Yaskawa INFORM job: N_R2_D100(P)(125,-90).JBI

/JOB
//NAME N_R2_D100(P)(125,-90)
//POS
///NPOS 515,515,515,27,0,0
///TOOL 0
///POSTYPE PULSE
///PULSE
C00000=15447,202281,164649,0,0,0
C00001=2000,202281,164649,0,0,0
C00002=24681,215512,219733,34338,41733,-28268
C00003=32295,212576,219732,43308,47198,-30665
C00004=90115,188704,203220,30079,59092,-18346
C00005=118922,140578,219095,27318,53560,2790
C00006=119744,138577,231841,24125,52341,6575
C00007=120497,123172,224477,21988,53305,9252
C00008=120847,115536,217515,22106,53618,9360
C00009=120990,112382,214541,22138,53803,9417
C00010=120986,108819,210345,21935,54503,9573
C00011=120990,112382,214541,22138,53803,9417
C00012=120993,109322,210918,21965,54414,9554
C00013=121006,109286,212535,22245,53471,9344
C00014=120993,109322,210918,21965,54414,9554
C00015=120850,112547,214017,21943,54191,9489
C00016=120501,120324,221241,21847,53796,9362
C00017=120536,123232,224555,-26557,40851,-26231
C00018=120886,115599,217598,-26179,41201,-26302
C00019=121030,112446,214627,-25996,41400,-26348
C00020=121025,108886,210434,-25635,42079,-26568
C00021=121030,112446,214627,-25996,41400,-26348
C00022=121027,109434,211061,-25684,41985,-26538
C00023=121040,109396,212675,-26172,41070,-26238
C00024=121027,109434,211061,-25684,41985,-26538
C00025=120883,112656,214154,-25882,41749,-26482
C00026=120533,120428,221368,-26294,41319,-26389
C00027=120975,122874,223899,-30521,46678,-26217
C00028=120979,115537,217604,-30470,46767,-26249
C00029=120981,112512,214915,-30422,46855,-26280
C00030=120976,108961,210733,-30079,47506,-26511
C00031=120981,112512,214915,-30422,46855,-26280
C00032=121048,109562,211421,-30089,47413,-26468
C00033=121062,109514,213024,-30551,46535,-26155
C00034=121048,109562,211421,-30089,47413,-26468
C00035=121046,112648,214220,-30153,47293,-26427
C00036=121040,120109,220750,-30241,47132,-26371
C00037=120918,149818,244976,-34417,46656,-25497
C00038=121562,167201,228013,-36113,61828,-28968
C00039=121102,161444,224515,-36573,61063,-28803
C00040=120915,159084,223008,-36750,60787,-28748
C00041=120912,155920,219969,-36672,60985,-28824
C00042=120915,159084,223008,-36750,60787,-28748
C00043=120918,156397,220402,-36676,60969,-28816
C00044=120925,157431,223143,-37055,60036,-28457
C00045=120918,156397,220402,-36676,60969,-28816
C00046=121105,158787,221971,-36508,61226,-28864
C00047=121564,164611,225614,-36067,61947,-29011
C00048=120584,167052,227666,-19839,59929,-30919
C00049=120814,161247,224144,-19904,59192,-30727
C00050=120908,158867,222626,-19923,58932,-30657
C00051=120905,155698,219577,-19875,59165,-30702
C00052=120908,158867,222626,-19923,58932,-30657
C00053=120916,156209,220066,-19878,59131,-30693
C00054=120923,157252,222817,-20111,58041,-30483
C00055=120916,156209,220066,-19878,59131,-30693
C00056=120822,158619,221647,-19864,59369,-30759
C00057=120592,164492,225315,-19810,60055,-30940
C00058=133732,167122,227890,29835,67104,20906
C00059=134129,161252,224225,30182,66361,20791
C00060=134290,158846,222649,30317,66097,20753
C00061=134272,155679,219605,30256,66314,20811
C00062=134290,158846,222649,30317,66097,20753
C00063=134298,156172,220059,30274,66286,20809
C00064=134507,157193,222762,30624,65256,20561
C00065=134298,156172,220059,30274,66286,20809
C00066=134137,158608,221700,30145,66529,20840
C00067=133740,164547,225513,29811,67224,20942
C00068=134000,188837,240725,29229,55891,39405
C00069=133801,188111,227982,27078,47780,60327
C00070=134153,183383,226108,27654,46559,60070
C00071=134296,181436,225266,27883,46096,59971
C00072=134279,178559,222861,27880,46101,59967
C00073=134296,181436,225266,27883,46096,59971
C00074=134291,178989,223219,27881,46099,59970
C00075=134475,180502,226338,28426,45044,59685
C00076=134291,178989,223219,27881,46099,59970
C00077=134148,180960,224110,27661,46546,60064
C00078=133797,185745,226100,27101,47729,60309
C00079=127590,202258,243387,866,47025,1941
C00080=121190,187961,227709,-25550,51120,-56262
C00081=120985,183329,226006,-26052,49870,-55982
C00082=120902,181420,225233,-26252,49395,-55874
C00083=120900,178540,222822,-26251,49398,-55875
C00084=120902,181420,225233,-26252,49395,-55874
C00085=120892,178980,223180,-26250,49401,-55879
C00086=120898,180522,226354,-26695,48358,-55570
C00087=120892,178980,223180,-26250,49401,-55879
C00088=120975,180912,224000,-26056,49860,-55983
C00089=121179,185599,225817,-25568,51072,-56253
C00090=121185,188297,228247,-25605,50975,-56224
C00091=120980,183661,226545,-26112,49722,-55942
C00092=120897,181750,225774,-26314,49247,-55833
C00093=120894,178874,223373,-26314,49246,-55833
C00094=120897,181750,225774,-26314,49247,-55833
C00095=120898,179301,223688,-26304,49270,-55839
C00096=120904,180831,226847,-26751,48230,-55529
C00097=120898,179301,223688,-26304,49270,-55839
C00098=120981,181234,224507,-26109,49730,-55943
C00099=121186,185925,226319,-25616,50945,-56215
C00100=123255,190595,236639,-58374,45131,30448
C00101=121545,184773,229975,-57949,45038,29555
C00102=120876,182366,227165,-57724,45033,29172
C00103=120874,179498,224782,-57730,45028,29175
C00104=120876,182366,227165,-57724,45033,29172
C00105=120862,179977,225120,-57701,45044,29152
C00106=120856,178398,221901,-56736,45697,28529
C00107=120862,179977,225120,-57701,45044,29152
C00108=121345,179993,223956,-56969,45650,28853
C00109=120328,180009,223979,-57246,45221,28671
C00110=121345,179993,223956,-56969,45650,28853
C00111=122010,182441,226833,-57205,45639,29244
C00112=123712,188347,233635,-57658,45697,30155
C00113=134995,214964,238467,-8691,44212,8832
C00114=134559,207525,231549,-8564,44604,8626
C00115=134389,204482,228633,-8506,44818,8540
C00116=134374,201971,226926,-8539,44580,8557
C00117=134389,204482,228633,-8506,44818,8540
C00118=134390,202551,227390,-8540,44593,8562
C00119=134223,200539,223898,-8355,45682,8396
C00120=134390,202551,227390,-8540,44593,8562
C00121=134560,205616,230359,-8602,44359,8650
C00122=134996,213102,237394,-8737,43918,8862
C00123=144287,210385,244112,-8132,41075,13860
C00124=162510,180487,234335,-6563,37802,23826
C00125=161591,173217,227359,-6507,38310,23477
C00126=161227,170231,224409,-6476,38572,23335
C00127=161244,167363,222022,-6476,38567,23341
C00128=161227,170231,224409,-6476,38572,23335
C00129=161271,168139,222752,-6483,38519,23354
C00130=160731,166668,219858,-6355,39511,23094
C00131=161271,168139,222752,-6483,38519,23354
C00132=161635,171154,225763,-6517,38235,23498
C00133=162555,178484,232873,-6581,37676,23852
C00134=147345,180992,237476,47268,20987,-11030
C00135=147676,173490,228422,44084,22107,-9407
C00136=147804,170370,224593,42795,22624,-8748
C00137=147814,167507,222218,42808,22614,-8751
C00138=147804,170370,224593,42795,22624,-8748
C00139=147835,168251,222850,42814,22602,-8748
C00140=147464,166660,219713,41151,23554,-8049
C00141=147835,168251,222850,42814,22602,-8748
C00142=147708,171402,226744,44147,22068,-9428
C00143=147378,178960,235933,47444,20911,-11105
C00144=133904,162048,228097,33647,50633,10192
C00145=127588,130671,218361,30951,63753,21604
C00146=128854,119558,220506,33838,57729,19894
C00147=129470,112494,214665,34247,57638,19934
C00148=129726,109579,212162,34397,57648,19967
C00149=129742,112224,215274,34604,57184,19801
C00150=129569,109596,210947,34036,58296,20180
C00151=132366,109517,211748,36018,57562,20250
C00152=135842,109408,211034,38109,57490,20655
C00153=138408,109303,210375,39617,57467,20980
C00154=138062,112231,212930,39423,57456,20929
C00155=137230,119317,218881,38897,57538,20855
C00156=115967,118809,218377,-25545,47752,-39219
C00157=116191,112195,213396,-25545,47467,-39108
C00158=116285,109468,211254,-25523,47399,-39076
C00159=116282,112131,214390,-25748,46891,-38928
C00160=116355,109459,210002,-25188,48101,-39267
C00161=118928,109470,211349,-24010,47549,-38784
C00162=122456,109452,211317,-21960,47808,-38412
C00163=125098,109423,211175,-20407,48050,-38145
C00164=124889,112154,213338,-20506,48104,-38183
C00165=124389,118775,218368,-20698,48360,-38302
C00166=123290,120857,220014,-35984,60052,-26242
C00167=122625,114409,215262,-36544,59662,-26177
C00168=122348,111754,213220,-36761,59545,-26166
C00169=122316,111747,211968,-36523,60163,-26407
C00170=122353,114378,216284,-36944,59111,-25997
C00171=119728,111769,213256,-38469,59242,-26369
C00172=117109,111771,213192,-40159,58971,-26586
C00173=123727,102355,205526,-46183,63931,-23649
C00174=124304,105056,207757,-45789,64016,-23616
C00175=125681,111582,212923,-44802,64320,-23585
C00176=122698,156476,234876,-36527,60349,-36905
C00177=122449,163722,222666,-33648,69836,-40138
C00178=121994,159688,221694,-34169,68496,-39820
C00179=121806,158013,221215,-34384,67981,-39697
C00180=121791,157173,219089,-34204,68709,-39940
C00181=121809,160369,223457,-34419,67841,-39650
C00182=120088,158037,221255,-35242,67579,-39982
C00183=118371,158016,221193,-36088,67201,-40276
C00184=122679,152032,219113,-44889,69211,-37700
C00185=123062,153728,219715,-44556,69677,-37816
C00186=123991,157822,220989,-43746,70895,-38125
C00187=117611,162371,222198,-19784,66538,-43060
C00188=117793,158216,221101,-19914,65186,-42779
C00189=117869,156493,220572,-19966,64669,-42670
C00190=117868,158864,222847,-19994,64498,-42639
C00191=117897,155666,218455,-19819,65501,-42813
C00192=119597,156527,220662,-19178,64861,-42329
C00193=121845,156504,220628,-18142,65154,-41894
C00194=123573,156435,220485,-17338,65412,-41565
C00195=123448,158166,221035,-17324,65925,-41671
C00196=123147,162343,222180,-17285,67268,-41941
C00197=130679,163960,225066,30363,74587,25346
C00198=131116,159105,222943,30757,73467,25136
C00199=131295,157106,221999,30917,73046,25058
C00200=131307,159462,224250,30949,72892,25018
C00201=131175,156320,219941,30731,73816,25246
C00202=133013,156803,221311,31804,72926,25408
C00203=135283,156324,220230,32955,72802,25889
C00204=136969,155906,219294,33795,72736,26262
C00205=136752,157909,220273,33612,73143,26338
C00206=136221,162768,222474,33163,74225,26543
C00207=131937,177942,231219,28739,51369,58836
C00208=131103,185328,225941,26199,57946,60545
C00209=131497,181762,225676,26766,56357,60246
C00210=131658,180274,225484,26999,55742,60128
C00211=131668,182419,227259,26999,55748,60133
C00212=131547,179118,223115,26715,56541,60311
C00213=133175,179856,224698,27300,55643,60570
C00214=135134,179225,223518,27660,55557,61158
C00215=136627,178672,222487,27910,55524,61620
C00216=136437,180155,222700,27670,56130,61731
C00217=135971,183707,223014,27083,57697,62015
C00218=123486,183308,222755,-21677,66267,-58163
C00219=123319,180552,223572,-22045,64449,-57850
C00220=123251,179379,223810,-22199,63739,-57726
C00221=123223,178175,221372,-22053,64554,-57898
C00222=123255,181534,225607,-22197,63742,-57725
C00223=121722,179460,223953,-22704,63409,-58082
C00224=119733,179485,223987,-23346,63019,-58556
C00225=118204,179443,223897,-23827,62749,-58927
C00226=118311,180627,223678,-23647,63452,-59052
C00227=118572,183412,222911,-23216,65258,-59366
C00228=122206,184212,222841,-27321,66765,-58270
C00229=121798,181549,223731,-27836,64961,-57929
C00230=121630,180415,223999,-28052,64257,-57793
C00231=121618,179195,221548,-27868,65037,-58001
C00232=121632,182559,225773,-28049,64266,-57795
C00233=120107,180439,224035,-28563,63890,-58140
C00234=118635,180411,223973,-29045,63559,-58483
C00235=122580,176867,224399,-39006,63999,-56229
C00236=122918,178040,224252,-38675,64647,-56380
C00237=123742,180810,223670,-37882,66314,-56760
C00238=125862,202189,241988,-26904,43300,-21160
C00239=128120,179057,235701,-24559,16531,13780
C00240=127696,171561,226511,-21973,18124,12452
C00241=127532,168433,222615,-20995,18834,11946
C00242=127606,170000,225314,-21985,18047,12432
C00243=127545,166519,221260,-21162,18697,12029
C00244=125920,168634,223016,-20023,18448,11037
C00245=112939,168466,222575,-9357,17147,2426
C00246=116539,165584,219262,-37323,21752,16959
C00247=116784,168723,223233,-38712,21158,17694
C00248=117416,176211,232564,-42212,19875,19542
C00249=121932,189645,236423,-2159,24410,9442
C00250=125769,180703,224227,31786,27614,1052
C00251=125876,172261,214331,30088,29100,1944
C00252=125917,168698,210066,29379,29784,2319
C00253=125917,170827,211817,29365,29798,2326
C00254=125970,170335,212982,30203,28938,1911
C00255=142087,161474,197407,20119,29855,11283
C00256=142171,165460,202283,20666,28944,11023
C00257=142389,174687,213323,21963,26983,10423
C00258=90115,188704,203220,30079,59092,-18346
C00259=32295,212576,219732,43308,47198,-30665
C00260=2000,202281,164649,0,0,0
C00261=15447,202281,164649,0,0,0
C00262=15447,202281,164649,0,0,0
C00263=15447,202281,164649,0,0,0
C00264=15447,202281,164649,0,0,0
C00265=-58673,196004,224446,-17944,28085,-14939
C00266=-145889,122722,224235,-48016,46095,-18882
C00267=-146704,115040,217017,-48175,46329,-19173
C00268=-147038,111863,213932,-48195,46466,-19322
C00269=-146989,108284,209714,-47640,46990,-19664
C00270=-147038,111863,213932,-48195,46466,-19322
C00271=-146995,108789,210290,-47709,46924,-19621
C00272=-147588,108743,211799,-48743,46197,-19229
C00273=-146995,108789,210290,-47709,46924,-19621
C00274=-146662,112041,213504,-47715,46759,-19455
C00275=-145849,119871,220993,-47617,46464,-19124
C00276=-145866,122721,224221,12828,42108,23463
C00277=-146680,115039,217002,12262,42622,23440
C00278=-147014,111862,213917,12020,42894,23437
C00279=-146965,108283,209699,11881,43634,23545
C00280=-147014,111862,213917,12020,42894,23437
C00281=-146966,108834,210330,11903,43530,23531
C00282=-147558,108787,211839,11788,42619,23332
C00283=-146966,108834,210330,11903,43530,23531
C00284=-146633,112084,213542,12150,43218,23530
C00285=-145821,119912,221027,12727,42616,23544
C00286=-99896,140771,234890,41057,43978,29210
C00287=-81385,119911,205689,47423,48192,34395
C00288=-80612,112172,198576,47559,48302,34669
C00289=-80295,108915,195463,47563,48400,34817
C00290=-80351,104656,190369,46930,49067,35225
C00291=-80295,108915,195463,47563,48400,34817
C00292=-80403,105399,191277,47016,48956,35141
C00293=-79657,105979,193427,48055,48085,34783
C00294=-80403,105399,191277,47016,48956,35141
C00295=-80719,108783,194591,47047,48817,34969
C00296=-81490,116767,202104,46988,48624,34642
C00297=-121434,148984,228686,40232,53743,25735
C00298=-121121,165984,226349,36450,61818,29263
C00299=-120652,160195,222770,36904,61078,29109
C00300=-120461,157820,221228,37078,60813,29058
C00301=-120460,154625,218133,36993,61025,29139
C00302=-120461,157820,221228,37078,60813,29058
C00303=-120466,155107,218575,36998,61007,29131
C00304=-120457,156175,221361,37390,60066,28768
C00305=-120466,155107,218575,36998,61007,29131
C00306=-120656,157514,220182,36833,61253,29174
C00307=-121124,163375,223912,36400,61948,29310
C00308=-120154,166157,226580,20192,59897,31174
C00309=-120372,160332,223012,20262,59178,30985
C00310=-120461,157943,221473,20283,58926,30916
C00311=-120460,154752,218385,20230,59171,30964
C00312=-120461,157943,221473,20283,58926,30916
C00313=-120471,155268,218880,20234,59135,30954
C00314=-120462,156328,221657,20479,58039,30743
C00315=-120471,155268,218880,20234,59135,30954
C00316=-120382,157688,220483,20218,59365,31019
C00317=-120164,163584,224201,20160,60032,31197
C00318=-146440,166394,227138,-35573,64457,-23044
C00319=-146979,160414,223226,-36008,63785,-22942
C00320=-147198,157963,221547,-36175,63549,-22912
C00321=-147166,154780,218475,-36088,63764,-22982
C00322=-147198,157963,221547,-36175,63549,-22912
C00323=-147192,155271,218924,-36107,63739,-22979
C00324=-147579,156256,221527,-36607,62756,-22717
C00325=-147192,155271,218924,-36107,63739,-22979
C00326=-146973,157755,220671,-35948,63955,-23001
C00327=-146435,163809,224737,-35531,64581,-23086
C00328=-120313,172340,242320,-34299,35799,-50864
C00329=-120152,166165,226604,-29898,41627,-53270
C00330=-120370,160336,223029,-30397,40891,-53053
C00331=-120459,157946,221489,-30580,40630,-52978
C00332=-120458,154754,218399,-30427,40857,-53068
C00333=-120459,157946,221489,-30580,40630,-52978
C00334=-120469,155236,218868,-30453,40819,-53057
C00335=-120460,156294,221642,-31149,39814,-52643
C00336=-120469,155236,218868,-30453,40819,-53057
C00337=-120380,157659,220474,-30285,41060,-53123
C00338=-120162,163559,224200,-29823,41748,-53319
C00339=-120808,166152,226594,30394,41466,53466
C00340=-120566,160321,223012,30904,40730,53252
C00341=-120468,157930,221468,31092,40469,53177
C00342=-120467,154738,218378,30936,40695,53270
C00343=-120468,157930,221468,31092,40469,53177
C00344=-120458,155231,218846,30958,40663,53260
C00345=-120449,156289,221621,31673,39660,52843
C00346=-120458,155231,218846,30958,40663,53260
C00347=-120556,157654,220455,30787,40904,53326
C00348=-120797,163556,224188,30312,41591,53519
C00349=-120791,196764,225758,23929,56035,57876
C00350=-120587,192763,224927,24383,54574,57590
C00351=-120504,191103,224507,24568,54012,57478
C00352=-120503,188374,222390,24597,53921,57455
C00353=-120504,191103,224507,24568,54012,57478
C00354=-120507,188771,222654,24584,53959,57464
C00355=-120500,190581,226050,24939,52900,57195
C00356=-120507,188771,222654,24584,53959,57464
C00357=-120590,190453,223116,24404,54508,57573
C00358=-120794,194507,224049,23958,55937,57852
C00359=-122901,177919,234113,63280,42164,-33162
C00360=-121117,172090,227052,62620,42118,-32100
C00361=-120421,169668,224067,62288,42131,-31644
C00362=-120420,166625,221312,62159,42195,-31566
C00363=-120421,169668,224067,62288,42131,-31644
C00364=-120408,167144,221724,62151,42197,-31556
C00365=-120417,165777,218657,61011,42789,-30863
C00366=-120408,167144,221724,62151,42197,-31556
C00367=-120925,167366,220808,61321,42738,-31237
C00368=-119855,167357,220784,61673,42315,-31065
C00369=-120925,167366,220808,61321,42738,-31237
C00370=-121617,169838,223867,61665,42707,-31701
C00371=-123392,175769,231085,62355,42716,-32781
C00372=-120775,202280,235367,5153,48165,-2931
C00373=-120574,194769,228526,5129,48504,-2846
C00374=-120495,191692,225634,5115,48698,-2809
C00375=-120494,188968,223530,5123,48593,-2814
C00376=-120495,191692,225634,5115,48698,-2809
C00377=-120503,189591,224082,5125,48574,-2818
C00378=-120509,187723,220613,5036,49745,-2759
C00379=-120503,189591,224082,5125,48574,-2818
C00380=-120581,192697,227036,5141,48357,-2856
C00381=-120782,200268,234015,5169,47964,-2945
C00382=-121097,206999,244193,5681,44142,-5775
C00383=-121079,191512,235492,5954,40481,-9245
C00384=-120657,183850,227977,5863,41145,-9051
C00385=-120492,180703,224799,5820,41473,-8971
C00386=-120490,178006,222744,5834,41353,-8978
C00387=-120492,180703,224799,5820,41473,-8971
C00388=-120494,178766,223429,5838,41322,-8982
C00389=-120501,176832,219899,5707,42495,-8905
C00390=-120494,178766,223429,5838,41322,-8982
C00391=-120660,181940,226664,5883,40972,-9064
C00392=-121082,189654,234305,5981,40258,-9262
C00393=-146775,180220,236645,-47419,21377,11449
C00394=-147132,172694,227537,-44253,22500,9822
C00395=-147271,169560,223681,-42968,23019,9160
C00396=-147281,166682,221276,-42964,23016,9155
C00397=-147271,169560,223681,-42968,23019,9160
C00398=-147302,167430,221917,-42975,23002,9154
C00399=-146946,165817,218742,-41312,23957,8448
C00400=-147302,167430,221917,-42975,23002,9154
C00401=-147164,170597,225840,-44303,22466,9837
C00402=-146807,178182,235087,-47582,21306,11517
C00403=-128844,167489,219119,15109,24995,-9484
C00404=-128455,158835,208529,13890,26957,-8768
C00405=-128304,155133,203914,13405,27852,-8482
C00406=-128303,157478,206048,13453,27746,-8505
C00407=-128377,156724,206863,13887,26890,-8745
C00408=-113473,155144,203864,7072,26584,-1170
C00409=-120204,149292,197389,35449,33024,-10735
C00410=-120464,153150,202294,36424,32253,-11330
C00411=-121134,162040,213399,38741,30633,-12744
C00412=-125965,166758,224416,9420,26881,-6319
C00413=-137280,145505,221527,-60849,19455,9531
C00414=-137453,137208,210771,-55362,20695,6872
C00415=-137521,133648,206098,-53143,21305,5791
C00416=-137716,135087,208858,-55194,20670,6709
C00417=-137560,131229,203824,-52823,21390,5626
C00418=-156550,123741,185060,-35830,21532,-8194
C00419=-156648,128309,191123,-37966,20387,-7202
C00420=-156899,138396,204316,-43383,18060,-4720
C00421=-117911,183564,223283,-22555,61467,-57170
C00422=-118076,180119,223191,-22961,59849,-56871
C00423=-118143,178678,223067,-23129,59222,-56752
C00424=-118172,177467,220617,-22939,60034,-56939
C00425=-118142,180842,224883,-23129,59217,-56751
C00426=-119670,178746,223204,-23560,58878,-57121
C00427=-121656,178756,223231,-24104,58472,-57611
C00428=-123183,178701,223135,-24507,58190,-57997
C00429=-123083,180153,223278,-24318,58813,-58115
C00430=-122836,183626,223419,-23858,60420,-58413
C00431=-123435,182649,222116,21854,66109,58333
C00432=-123257,179876,222901,22228,64300,58022
C00433=-123184,178696,223127,22385,63595,57898
C00434=-123187,180861,224942,22385,63591,57896
C00435=-123163,177487,220678,22234,64413,58071
C00436=-121656,178751,223223,22883,63276,58258
C00437=-119670,178742,223197,23516,62901,58735
C00438=-118143,178673,223059,23990,62643,59110
C00439=-118255,179863,222853,23808,63343,59234
C00440=-118526,182662,222117,23372,65138,59545
C00441=-122155,183298,221760,27476,66700,58464
C00442=-121736,180626,222622,27994,64905,58126
C00443=-121564,179487,222878,28211,64206,57992
C00444=-121566,181643,224676,28211,64207,57992
C00445=-121559,178253,220406,28022,64992,58201
C00446=-120046,179485,222867,28713,63850,58342
C00447=-118578,179431,222759,29186,63530,58689
C00448=-122506,175989,223283,39187,63899,56423
C00449=-122848,177168,223153,38856,64543,56572
C00450=-123680,179952,222608,38062,66198,56948
C00451=-122755,177840,230233,35129,68690,45019
C00452=-122402,163008,221792,33920,69743,40290
C00453=-121935,158958,220781,34447,68416,39976
C00454=-121743,157277,220286,34663,67908,39855
C00455=-121745,159644,222551,34701,67761,39805
C00456=-121735,156426,218144,34477,68638,40099
C00457=-120029,157280,220283,35512,67514,40144
C00458=-118316,157238,220178,36348,67145,40443
C00459=-122598,151300,218166,45203,69096,37849
C00460=-122985,153006,218789,44869,69556,37963
C00461=-123926,157123,220115,44056,70760,38266
C00462=-117568,161718,221460,20034,66474,43214
C00463=-117738,157551,220337,20172,65132,42934
C00464=-117808,155823,219795,20227,64620,42826
C00465=-117844,154989,217669,20075,65454,42969
C00466=-117806,158204,222092,20257,64441,42793
C00467=-119533,155877,219929,19446,64800,42481
C00468=-121779,155880,219951,18418,65078,42043
C00469=-123506,155832,219850,17618,65325,41711
C00470=-123387,157569,220410,17601,65834,41816
C00471=-123098,161760,221582,17552,67167,42086
C00472=-130606,163214,224103,-30003,74848,-25248
C00473=-131030,158350,221955,-30383,73737,-25043
C00474=-131204,156346,220999,-30538,73320,-24967
C00475=-131091,155548,218923,-30359,74095,-25155
C00476=-131214,158715,223275,-30570,73159,-24925
C00477=-132920,156060,220349,-31425,73190,-25315
C00478=-135189,155602,219317,-32580,73054,-25793
C00479=-136875,155200,218418,-33422,72979,-26163
C00480=-136662,157207,219408,-33245,73383,-26236
C00481=-136144,162078,221634,-32808,74457,-26438
C00482=-132038,149022,237746,-34581,60859,-21400
C00483=-128805,119167,220009,-33427,57827,-19835
C00484=-129404,112081,214130,-33821,57749,-19877
C00485=-129653,109155,211609,-33965,57764,-19912
C00486=-129507,109170,210390,-33615,58415,-20122
C00487=-129667,111811,214741,-34170,57293,-19745
C00488=-132294,109098,211223,-35589,57668,-20192
C00489=-135774,108996,210545,-37688,57583,-20592
C00490=-138345,108896,209914,-39203,57551,-20915
C00491=-138006,111834,212485,-39015,57535,-20863
C00492=-137190,118943,218472,-38505,57606,-20785
C00493=-115927,118422,217977,25886,47656,39303
C00494=-116133,111786,212957,25894,47383,39196
C00495=-116219,109048,210797,25875,47320,39167
C00496=-116300,109040,209546,25530,48020,39359
C00497=-116214,111722,213951,26107,46807,39015
C00498=-118862,109058,210922,24371,47459,38870
C00499=-122393,109050,210931,22328,47705,38493
C00500=-125039,109027,210818,20779,47936,38222
C00501=-124837,111767,212997,20874,47986,38258
C00502=-124356,118411,218064,21058,48232,38374
C00503=-123256,120475,219528,36367,59980,26317
C00504=-122574,114004,214729,36934,59603,26258
C00505=-122288,111339,212667,37153,59490,26250
C00506=-122292,113975,215750,37342,59054,26077
C00507=-122268,111330,211411,36904,60107,26492
C00508=-119672,111348,212674,38852,59194,26458
C00509=-117058,111342,212580,40530,58930,26680
C00510=-123636,101884,204901,46615,63860,23731
C00511=-124221,104599,207161,46219,63940,23693
C00512=-125617,111156,212391,45228,64231,23652
C00513=-58673,196004,224446,-17944,28085,-14939
C00514=15447,202281,164649,0,0,0
BC00000=0,675528,1075229
BC00001=0,1249520,1075229
BC00002=20074,1273230,1075229
BC00003=22843,1276500,1075229
BC00004=181219,1349640,881743
BC00005=259614,1271622,997019
BC00006=263455,1253369,961473
BC00007=265649,1242939,941161
BC00008=265649,1242939,941161
BC00009=265649,1242939,941161
BC00010=265649,1242939,941161
BC00011=265649,1242939,941161
BC00012=265649,1242939,941161
BC00013=265649,1242939,941161
BC00014=265649,1242939,941161
BC00015=265649,1242939,941161
BC00016=265649,1242939,941161
BC00017=279094,1259762,979345
BC00018=279094,1259762,979345
BC00019=279094,1259762,979345
BC00020=279094,1259762,979345
BC00021=279094,1259762,979345
BC00022=279094,1259762,979345
BC00023=279094,1259762,979345
BC00024=279094,1259762,979345
BC00025=279094,1259762,979345
BC00026=279094,1259762,979345
BC00027=338482,1253298,958814
BC00028=338482,1253298,958814
BC00029=338482,1253298,958814
BC00030=338482,1253298,958814
BC00031=338482,1253298,958814
BC00032=338482,1253298,958814
BC00033=338482,1253298,958814
BC00034=338482,1253298,958814
BC00035=338482,1253298,958814
BC00036=338482,1253298,958814
BC00037=333821,1266832,919202
BC00038=321005,1304050,810268
BC00039=321005,1304050,810268
BC00040=321005,1304050,810268
BC00041=321005,1304050,810268
BC00042=321005,1304050,810268
BC00043=321005,1304050,810268
BC00044=321005,1304050,810268
BC00045=321005,1304050,810268
BC00046=321005,1304050,810268
BC00047=321005,1304050,810268
BC00048=279090,1297669,836196
BC00049=279090,1297669,836196
BC00050=279090,1297669,836196
BC00051=279090,1297669,836196
BC00052=279090,1297669,836196
BC00053=279090,1297669,836196
BC00054=279090,1297669,836196
BC00055=279090,1297669,836196
BC00056=279090,1297669,836196
BC00057=279090,1297669,836196
BC00058=308990,1283728,803935
BC00059=308990,1283728,803935
BC00060=308990,1283728,803935
BC00061=308990,1283728,803935
BC00062=308990,1283728,803935
BC00063=308990,1283728,803935
BC00064=308990,1283728,803935
BC00065=308990,1283728,803935
BC00066=308990,1283728,803935
BC00067=308990,1283728,803935
BC00068=309388,1296619,799441
BC00069=309813,1310369,794648
BC00070=309813,1310369,794648
BC00071=309813,1310369,794648
BC00072=309813,1310369,794648
BC00073=309813,1310369,794648
BC00074=309813,1310369,794648
BC00075=309813,1310369,794648
BC00076=309813,1310369,794648
BC00077=309813,1310369,794648
BC00078=309813,1310369,794648
BC00079=290509,1311906,794287
BC00080=271204,1313444,793926
BC00081=271204,1313444,793926
BC00082=271204,1313444,793926
BC00083=271204,1313444,793926
BC00084=271204,1313444,793926
BC00085=271204,1313444,793926
BC00086=271204,1313444,793926
BC00087=271204,1313444,793926
BC00088=271204,1313444,793926
BC00089=271204,1313444,793926
BC00090=339752,1313535,794120
BC00091=339752,1313535,794120
BC00092=339752,1313535,794120
BC00093=339752,1313535,794120
BC00094=339752,1313535,794120
BC00095=339752,1313535,794120
BC00096=339752,1313535,794120
BC00097=339752,1313535,794120
BC00098=339752,1313535,794120
BC00099=339752,1313535,794120
BC00100=309596,1336055,723788
BC00101=309596,1336055,723788
BC00102=309596,1336055,723788
BC00103=309596,1336055,723788
BC00104=309596,1336055,723788
BC00105=309596,1336055,723788
BC00106=309596,1336055,723788
BC00107=309596,1336055,723788
BC00108=309596,1336055,723788
BC00109=309596,1336055,723788
BC00110=309596,1336055,723788
BC00111=309596,1336055,723788
BC00112=309596,1336055,723788
BC00113=366840,1349942,659049
BC00114=366840,1349942,659049
BC00115=366840,1349942,659049
BC00116=366840,1349942,659049
BC00117=366840,1349942,659049
BC00118=366840,1349942,659049
BC00119=366840,1349942,659049
BC00120=366840,1349942,659049
BC00121=366840,1349942,659049
BC00122=366840,1349942,659049
BC00123=369598,1321086,746352
BC00124=375224,1262220,924452
BC00125=375224,1262220,924452
BC00126=375224,1262220,924452
BC00127=375224,1262220,924452
BC00128=375224,1262220,924452
BC00129=375224,1262220,924452
BC00130=375224,1262220,924452
BC00131=375224,1262220,924452
BC00132=375224,1262220,924452
BC00133=375224,1262220,924452
BC00134=339925,1300732,881743
BC00135=339925,1300732,881743
BC00136=339925,1300732,881743
BC00137=339925,1300732,881743
BC00138=339925,1300732,881743
BC00139=339925,1300732,881743
BC00140=339925,1300732,881743
BC00141=339925,1300732,881743
BC00142=339925,1300732,881743
BC00143=339925,1300732,881743
BC00144=315652,1292340,901479
BC00145=299654,1262212,953023
BC00146=298993,1238691,912276
BC00147=298993,1238691,912276
BC00148=298993,1238691,912276
BC00149=298993,1238691,912276
BC00150=298993,1238691,912276
BC00151=298993,1238691,912276
BC00152=298993,1238691,912276
BC00153=298993,1238691,912276
BC00154=298993,1238691,912276
BC00155=298993,1238691,912276
BC00156=278815,1248832,951478
BC00157=278815,1248832,951478
BC00158=278815,1248832,951478
BC00159=278815,1248832,951478
BC00160=278815,1248832,951478
BC00161=278815,1248832,951478
BC00162=278815,1248832,951478
BC00163=278815,1248832,951478
BC00164=278815,1248832,951478
BC00165=278815,1248832,951478
BC00166=314804,1246682,892728
BC00167=314804,1246682,892728
BC00168=314804,1246682,892728
BC00169=314804,1246682,892728
BC00170=314804,1246682,892728
BC00171=314804,1246682,892728
BC00172=314804,1246682,892728
BC00173=314804,1246682,892728
BC00174=314804,1246682,892728
BC00175=314804,1246682,892728
BC00176=314801,1292959,892910
BC00177=314719,1294052,772836
BC00178=314719,1294052,772836
BC00179=314719,1294052,772836
BC00180=314719,1294052,772836
BC00181=314719,1294052,772836
BC00182=314719,1294052,772836
BC00183=314719,1294052,772836
BC00184=314719,1294052,772836
BC00185=314719,1294052,772836
BC00186=314719,1294052,772836
BC00187=278878,1286739,810029
BC00188=278878,1286739,810029
BC00189=278878,1286739,810029
BC00190=278878,1286739,810029
BC00191=278878,1286739,810029
BC00192=278878,1286739,810029
BC00193=278878,1286739,810029
BC00194=278878,1286739,810029
BC00195=278878,1286739,810029
BC00196=278878,1286739,810029
BC00197=311908,1275469,768683
BC00198=311908,1275469,768683
BC00199=311908,1275469,768683
BC00200=311908,1275469,768683
BC00201=311908,1275469,768683
BC00202=311908,1275469,768683
BC00203=311908,1275469,768683
BC00204=311908,1275469,768683
BC00205=311908,1275469,768683
BC00206=311908,1275469,768683
BC00207=311248,1293583,920117
BC00208=310634,1294320,778613
BC00209=310634,1294320,778613
BC00210=310634,1294320,778613
BC00211=310634,1294320,778613
BC00212=310634,1294320,778613
BC00213=310634,1294320,778613
BC00214=310634,1294320,778613
BC00215=310634,1294320,778613
BC00216=310634,1294320,778613
BC00217=310634,1294320,778613
BC00218=269571,1288878,766650
BC00219=269571,1288878,766650
BC00220=269571,1288878,766650
BC00221=269571,1288878,766650
BC00222=269571,1288878,766650
BC00223=269571,1288878,766650
BC00224=269571,1288878,766650
BC00225=269571,1288878,766650
BC00226=269571,1288878,766650
BC00227=269571,1288878,766650
BC00228=324029,1292263,751538
BC00229=324029,1292263,751538
BC00230=324029,1292263,751538
BC00231=324029,1292263,751538
BC00232=324029,1292263,751538
BC00233=324029,1292263,751538
BC00234=324029,1292263,751538
BC00235=324029,1292263,751538
BC00236=324029,1292263,751538
BC00237=324029,1292263,751538
BC00238=331457,1324273,767907
BC00239=337552,1339765,848258
BC00240=337552,1339765,848258
BC00241=337552,1339765,848258
BC00242=337552,1339765,848258
BC00243=337552,1339765,848258
BC00244=337552,1339765,848258
BC00245=337552,1339765,848258
BC00246=337552,1339765,848258
BC00247=337552,1339765,848258
BC00248=337552,1339765,848258
BC00249=326395,1340304,844891
BC00250=315775,1339017,839253
BC00251=315775,1339017,839253
BC00252=315775,1339017,839253
BC00253=315775,1339017,839253
BC00254=315775,1339017,839253
BC00255=315775,1339017,839253
BC00256=315775,1339017,839253
BC00257=315775,1339017,839253
BC00258=181219,1349640,881743
BC00259=22843,1276500,1075229
BC00260=0,1249520,1075229
BC00261=0,675528,1075229
BC00262=0,675528,1075229
BC00263=0,675528,1075229
BC00264=0,675528,1075229
BC00265=138607,763027,1056836
BC00266=322510,879121,952026
BC00267=322510,879121,952026
BC00268=322510,879121,952026
BC00269=322510,879121,952026
BC00270=322510,879121,952026
BC00271=322510,879121,952026
BC00272=322510,879121,952026
BC00273=322510,879121,952026
BC00274=322510,879121,952026
BC00275=322510,879121,952026
BC00276=326477,871688,980713
BC00277=326477,871688,980713
BC00278=326477,871688,980713
BC00279=326477,871688,980713
BC00280=326477,871688,980713
BC00281=326477,871688,980713
BC00282=326477,871688,980713
BC00283=326477,871688,980713
BC00284=326477,871688,980713
BC00285=326477,871688,980713
BC00286=267497,855485,958441
BC00287=255081,864777,953752
BC00288=255081,864777,953752
BC00289=255081,864777,953752
BC00290=255081,864777,953752
BC00291=255081,864777,953752
BC00292=255081,864777,953752
BC00293=255081,864777,953752
BC00294=255081,864777,953752
BC00295=255081,864777,953752
BC00296=255081,864777,953752
BC00297=320924,819371,961652
BC00298=320924,819371,812233
BC00299=320924,819371,812233
BC00300=320924,819371,812233
BC00301=320924,819371,812233
BC00302=320924,819371,812233
BC00303=320924,819371,812233
BC00304=320924,819371,812233
BC00305=320924,819371,812233
BC00306=320924,819371,812233
BC00307=320924,819371,812233
BC00308=278908,825639,838037
BC00309=278908,825639,838037
BC00310=278908,825639,838037
BC00311=278908,825639,838037
BC00312=278908,825639,838037
BC00313=278908,825639,838037
BC00314=278908,825639,838037
BC00315=278908,825639,838037
BC00316=278908,825639,838037
BC00317=278908,825639,838037
BC00318=344258,850073,804397
BC00319=344258,850073,804397
BC00320=344258,850073,804397
BC00321=344258,850073,804397
BC00322=344258,850073,804397
BC00323=344258,850073,804397
BC00324=344258,850073,804397
BC00325=344258,850073,804397
BC00326=344258,850073,804397
BC00327=344258,850073,804397
BC00328=268540,837164,928608
BC00329=268540,837164,928608
BC00330=268540,837164,928608
BC00331=268540,837164,928608
BC00332=268540,837164,928608
BC00333=268540,837164,928608
BC00334=268540,837164,928608
BC00335=268540,837164,928608
BC00336=268540,837164,928608
BC00337=268540,837164,928608
BC00338=268540,837164,928608
BC00339=271645,836699,929417
BC00340=271645,836699,929417
BC00341=271645,836699,929417
BC00342=271645,836699,929417
BC00343=271645,836699,929417
BC00344=271645,836699,929417
BC00345=271645,836699,929417
BC00346=271645,836699,929417
BC00347=271645,836699,929417
BC00348=271645,836699,929417
BC00349=340192,799254,723936
BC00350=340192,799254,723936
BC00351=340192,799254,723936
BC00352=340192,799254,723936
BC00353=340192,799254,723936
BC00354=340192,799254,723936
BC00355=340192,799254,723936
BC00356=340192,799254,723936
BC00357=340192,799254,723936
BC00358=340192,799254,723936
BC00359=309001,800829,792422
BC00360=309001,800829,792422
BC00361=309001,800829,792422
BC00362=309001,800829,792422
BC00363=309001,800829,792422
BC00364=309001,800829,792422
BC00365=309001,800829,792422
BC00366=309001,800829,792422
BC00367=309001,800829,792422
BC00368=309001,800829,792422
BC00369=309001,800829,792422
BC00370=309001,800829,792422
BC00371=309001,800829,792422
BC00372=321646,797982,745635
BC00373=321646,797982,745635
BC00374=321646,797982,745635
BC00375=321646,797982,745635
BC00376=321646,797982,745635
BC00377=321646,797982,745635
BC00378=321646,797982,745635
BC00379=321646,797982,745635
BC00380=321646,797982,745635
BC00381=321646,797982,745635
BC00382=296475,807012,791430
BC00383=260705,819844,856508
BC00384=260705,819844,856508
BC00385=260705,819844,856508
BC00386=260705,819844,856508
BC00387=260705,819844,856508
BC00388=260705,819844,856508
BC00389=260705,819844,856508
BC00390=260705,819844,856508
BC00391=260705,819844,856508
BC00392=260705,819844,856508
BC00393=339123,823007,883432
BC00394=339123,823007,883432
BC00395=339123,823007,883432
BC00396=339123,823007,883432
BC00397=339123,823007,883432
BC00398=339123,823007,883432
BC00399=339123,823007,883432
BC00400=339123,823007,883432
BC00401=339123,823007,883432
BC00402=339123,823007,883432
BC00403=340871,798500,921000
BC00404=340871,798500,921000
BC00405=340871,798500,921000
BC00406=340871,798500,921000
BC00407=340871,798500,921000
BC00408=340871,798500,921000
BC00409=340871,798500,921000
BC00410=340871,798500,921000
BC00411=340871,798500,921000
BC00412=343473,807454,949850
BC00413=352115,833503,1009314
BC00414=352115,833503,1009314
BC00415=352115,833503,1009314
BC00416=352115,833503,1009314
BC00417=352115,833503,1009314
BC00418=352115,833503,1009314
BC00419=352115,833503,1009314
BC00420=352115,833503,1009314
BC00421=270260,826762,778340
BC00422=270260,826762,778340
BC00423=270260,826762,778340
BC00424=270260,826762,778340
BC00425=270260,826762,778340
BC00426=270260,826762,778340
BC00427=270260,826762,778340
BC00428=270260,826762,778340
BC00429=270260,826762,778340
BC00430=270260,826762,778340
BC00431=270830,834917,768745
BC00432=270830,834917,768745
BC00433=270830,834917,768745
BC00434=270830,834917,768745
BC00435=270830,834917,768745
BC00436=270830,834917,768745
BC00437=270830,834917,768745
BC00438=270830,834917,768745
BC00439=270830,834917,768745
BC00440=270830,834917,768745
BC00441=325301,832050,753660
BC00442=325301,832050,753660
BC00443=325301,832050,753660
BC00444=325301,832050,753660
BC00445=325301,832050,753660
BC00446=325301,832050,753660
BC00447=325301,832050,753660
BC00448=325301,832050,753660
BC00449=325301,832050,753660
BC00450=325301,832050,753660
BC00451=317689,831131,771467
BC00452=315834,830096,774743
BC00453=315834,830096,774743
BC00454=315834,830096,774743
BC00455=315834,830096,774743
BC00456=315834,830096,774743
BC00457=315834,830096,774743
BC00458=315834,830096,774743
BC00459=315834,830096,774743
BC00460=315834,830096,774743
BC00461=315834,830096,774743
BC00462=279937,837039,812006
BC00463=279937,837039,812006
BC00464=279937,837039,812006
BC00465=279937,837039,812006
BC00466=279937,837039,812006
BC00467=279937,837039,812006
BC00468=279937,837039,812006
BC00469=279937,837039,812006
BC00470=279937,837039,812006
BC00471=279937,837039,812006
BC00472=312368,849486,768314
BC00473=312368,849486,768314
BC00474=312368,849486,768314
BC00475=312368,849486,768314
BC00476=312368,849486,768314
BC00477=312368,849486,768314
BC00478=312368,849486,768314
BC00479=312368,849486,768314
BC00480=312368,849486,768314
BC00481=312368,849486,768314
BC00482=304168,872987,860177
BC00483=299744,886342,911434
BC00484=299744,886342,911434
BC00485=299744,886342,911434
BC00486=299744,886342,911434
BC00487=299744,886342,911434
BC00488=299744,886342,911434
BC00489=299744,886342,911434
BC00490=299744,886342,911434
BC00491=299744,886342,911434
BC00492=299744,886342,911434
BC00493=280164,875026,952983
BC00494=280164,875026,952983
BC00495=280164,875026,952983
BC00496=280164,875026,952983
BC00497=280164,875026,952983
BC00498=280164,875026,952983
BC00499=280164,875026,952983
BC00500=280164,875026,952983
BC00501=280164,875026,952983
BC00502=280164,875026,952983
BC00503=315859,877538,894138
BC00504=315859,877538,894138
BC00505=315859,877538,894138
BC00506=315859,877538,894138
BC00507=315859,877538,894138
BC00508=315859,877538,894138
BC00509=315859,877538,894138
BC00510=315859,877538,894138
BC00511=315859,877538,894138
BC00512=315859,877538,894138
BC00513=138607,763027,1056836
BC00514=0,675528,1075229
EC00000=1108551,-556475
EC00001=1108551,-556475
EC00002=1108551,-556475
EC00003=1108551,-556475
EC00004=1108551,-556475
EC00005=1108551,-556475
EC00006=1108551,-556475
EC00007=1108551,-556475
EC00008=1108551,-556475
EC00009=1108551,-556475
EC00010=1108551,-556475
EC00011=1108551,-556475
EC00012=1108551,-556475
EC00013=1108551,-556475
EC00014=1108551,-556475
EC00015=1108551,-556475
EC00016=1108551,-556475
EC00017=1108551,-556475
EC00018=1108551,-556475
EC00019=1108551,-556475
EC00020=1108551,-556475
EC00021=1108551,-556475
EC00022=1108551,-556475
EC00023=1108551,-556475
EC00024=1108551,-556475
EC00025=1108551,-556475
EC00026=1108551,-556475
EC00027=1108551,-556475
EC00028=1108551,-556475
EC00029=1108551,-556475
EC00030=1108551,-556475
EC00031=1108551,-556475
EC00032=1108551,-556475
EC00033=1108551,-556475
EC00034=1108551,-556475
EC00035=1108551,-556475
EC00036=1108551,-556475
EC00037=1108551,-556475
EC00038=1108551,-556475
EC00039=1108551,-556475
EC00040=1108551,-556475
EC00041=1108551,-556475
EC00042=1108551,-556475
EC00043=1108551,-556475
EC00044=1108551,-556475
EC00045=1108551,-556475
EC00046=1108551,-556475
EC00047=1108551,-556475
EC00048=1108551,-556475
EC00049=1108551,-556475
EC00050=1108551,-556475
EC00051=1108551,-556475
EC00052=1108551,-556475
EC00053=1108551,-556475
EC00054=1108551,-556475
EC00055=1108551,-556475
EC00056=1108551,-556475
EC00057=1108551,-556475
EC00058=1108551,-556475
EC00059=1108551,-556475
EC00060=1108551,-556475
EC00061=1108551,-556475
EC00062=1108551,-556475
EC00063=1108551,-556475
EC00064=1108551,-556475
EC00065=1108551,-556475
EC00066=1108551,-556475
EC00067=1108551,-556475
EC00068=1108551,-556475
EC00069=1108551,-556475
EC00070=1108551,-556475
EC00071=1108551,-556475
EC00072=1108551,-556475
EC00073=1108551,-556475
EC00074=1108551,-556475
EC00075=1108551,-556475
EC00076=1108551,-556475
EC00077=1108551,-556475
EC00078=1108551,-556475
EC00079=1108551,-556475
EC00080=1108551,-556475
EC00081=1108551,-556475
EC00082=1108551,-556475
EC00083=1108551,-556475
EC00084=1108551,-556475
EC00085=1108551,-556475
EC00086=1108551,-556475
EC00087=1108551,-556475
EC00088=1108551,-556475
EC00089=1108551,-556475
EC00090=1108551,-556475
EC00091=1108551,-556475
EC00092=1108551,-556475
EC00093=1108551,-556475
EC00094=1108551,-556475
EC00095=1108551,-556475
EC00096=1108551,-556475
EC00097=1108551,-556475
EC00098=1108551,-556475
EC00099=1108551,-556475
EC00100=1108551,-556475
EC00101=1108551,-556475
EC00102=1108551,-556475
EC00103=1108551,-556475
EC00104=1108551,-556475
EC00105=1108551,-556475
EC00106=1108551,-556475
EC00107=1108551,-556475
EC00108=1108551,-556475
EC00109=1108551,-556475
EC00110=1108551,-556475
EC00111=1108551,-556475
EC00112=1108551,-556475
EC00113=1108551,-556475
EC00114=1108551,-556475
EC00115=1108551,-556475
EC00116=1108551,-556475
EC00117=1108551,-556475
EC00118=1108551,-556475
EC00119=1108551,-556475
EC00120=1108551,-556475
EC00121=1108551,-556475
EC00122=1108551,-556475
EC00123=1108551,-556475
EC00124=1108551,-556475
EC00125=1108551,-556475
EC00126=1108551,-556475
EC00127=1108551,-556475
EC00128=1108551,-556475
EC00129=1108551,-556475
EC00130=1108551,-556475
EC00131=1108551,-556475
EC00132=1108551,-556475
EC00133=1108551,-556475
EC00134=1108551,-556475
EC00135=1108551,-556475
EC00136=1108551,-556475
EC00137=1108551,-556475
EC00138=1108551,-556475
EC00139=1108551,-556475
EC00140=1108551,-556475
EC00141=1108551,-556475
EC00142=1108551,-556475
EC00143=1108551,-556475
EC00144=1108551,-556475
EC00145=1108551,-556475
EC00146=1108551,-556475
EC00147=1108551,-556475
EC00148=1108551,-556475
EC00149=1108551,-556475
EC00150=1108551,-556475
EC00151=1108551,-556475
EC00152=1108551,-556475
EC00153=1108551,-556475
EC00154=1108551,-556475
EC00155=1108551,-556475
EC00156=1108551,-556475
EC00157=1108551,-556475
EC00158=1108551,-556475
EC00159=1108551,-556475
EC00160=1108551,-556475
EC00161=1108551,-556475
EC00162=1108551,-556475
EC00163=1108551,-556475
EC00164=1108551,-556475
EC00165=1108551,-556475
EC00166=1108551,-556475
EC00167=1108551,-556475
EC00168=1108551,-556475
EC00169=1108551,-556475
EC00170=1108551,-556475
EC00171=1108551,-556475
EC00172=1108551,-556475
EC00173=1108551,-556475
EC00174=1108551,-556475
EC00175=1108551,-556475
EC00176=1108551,-556475
EC00177=1108551,-556475
EC00178=1108551,-556475
EC00179=1108551,-556475
EC00180=1108551,-556475
EC00181=1108551,-556475
EC00182=1108551,-556475
EC00183=1108551,-556475
EC00184=1108551,-556475
EC00185=1108551,-556475
EC00186=1108551,-556475
EC00187=1108551,-556475
EC00188=1108551,-556475
EC00189=1108551,-556475
EC00190=1108551,-556475
EC00191=1108551,-556475
EC00192=1108551,-556475
EC00193=1108551,-556475
EC00194=1108551,-556475
EC00195=1108551,-556475
EC00196=1108551,-556475
EC00197=1108551,-556475
EC00198=1108551,-556475
EC00199=1108551,-556475
EC00200=1108551,-556475
EC00201=1108551,-556475
EC00202=1108551,-556475
EC00203=1108551,-556475
EC00204=1108551,-556475
EC00205=1108551,-556475
EC00206=1108551,-556475
EC00207=1108551,-556475
EC00208=1108551,-556475
EC00209=1108551,-556475
EC00210=1108551,-556475
EC00211=1108551,-556475
EC00212=1108551,-556475
EC00213=1108551,-556475
EC00214=1108551,-556475
EC00215=1108551,-556475
EC00216=1108551,-556475
EC00217=1108551,-556475
EC00218=1108551,-556475
EC00219=1108551,-556475
EC00220=1108551,-556475
EC00221=1108551,-556475
EC00222=1108551,-556475
EC00223=1108551,-556475
EC00224=1108551,-556475
EC00225=1108551,-556475
EC00226=1108551,-556475
EC00227=1108551,-556475
EC00228=1108551,-556475
EC00229=1108551,-556475
EC00230=1108551,-556475
EC00231=1108551,-556475
EC00232=1108551,-556475
EC00233=1108551,-556475
EC00234=1108551,-556475
EC00235=1108551,-556475
EC00236=1108551,-556475
EC00237=1108551,-556475
EC00238=1108551,-556475
EC00239=1108551,-556475
EC00240=1108551,-556475
EC00241=1108551,-556475
EC00242=1108551,-556475
EC00243=1108551,-556475
EC00244=1108551,-556475
EC00245=1108551,-556475
EC00246=1108551,-556475
EC00247=1108551,-556475
EC00248=1108551,-556475
EC00249=1108551,-556475
EC00250=1108551,-556475
EC00251=1108551,-556475
EC00252=1108551,-556475
EC00253=1108551,-556475
EC00254=1108551,-556475
EC00255=1108551,-556475
EC00256=1108551,-556475
EC00257=1108551,-556475
EC00258=1108551,-556475
EC00259=1108551,-556475
EC00260=1108551,-556475
EC00261=1108551,-556475
EC00262=266052,-556475
EC00263=-266052,556475
EC00264=-1108551,556475
EC00265=-1108551,556475
EC00266=-1108551,556475
EC00267=-1108551,556475
EC00268=-1108551,556475
EC00269=-1108551,556475
EC00270=-1108551,556475
EC00271=-1108551,556475
EC00272=-1108551,556475
EC00273=-1108551,556475
EC00274=-1108551,556475
EC00275=-1108551,556475
EC00276=-1108551,556475
EC00277=-1108551,556475
EC00278=-1108551,556475
EC00279=-1108551,556475
EC00280=-1108551,556475
EC00281=-1108551,556475
EC00282=-1108551,556475
EC00283=-1108551,556475
EC00284=-1108551,556475
EC00285=-1108551,556475
EC00286=-1108551,556475
EC00287=-1108551,556475
EC00288=-1108551,556475
EC00289=-1108551,556475
EC00290=-1108551,556475
EC00291=-1108551,556475
EC00292=-1108551,556475
EC00293=-1108551,556475
EC00294=-1108551,556475
EC00295=-1108551,556475
EC00296=-1108551,556475
EC00297=-1108551,556475
EC00298=-1108551,556475
EC00299=-1108551,556475
EC00300=-1108551,556475
EC00301=-1108551,556475
EC00302=-1108551,556475
EC00303=-1108551,556475
EC00304=-1108551,556475
EC00305=-1108551,556475
EC00306=-1108551,556475
EC00307=-1108551,556475
EC00308=-1108551,556475
EC00309=-1108551,556475
EC00310=-1108551,556475
EC00311=-1108551,556475
EC00312=-1108551,556475
EC00313=-1108551,556475
EC00314=-1108551,556475
EC00315=-1108551,556475
EC00316=-1108551,556475
EC00317=-1108551,556475
EC00318=-1108551,556475
EC00319=-1108551,556475
EC00320=-1108551,556475
EC00321=-1108551,556475
EC00322=-1108551,556475
EC00323=-1108551,556475
EC00324=-1108551,556475
EC00325=-1108551,556475
EC00326=-1108551,556475
EC00327=-1108551,556475
EC00328=-1108551,556475
EC00329=-1108551,556475
EC00330=-1108551,556475
EC00331=-1108551,556475
EC00332=-1108551,556475
EC00333=-1108551,556475
EC00334=-1108551,556475
EC00335=-1108551,556475
EC00336=-1108551,556475
EC00337=-1108551,556475
EC00338=-1108551,556475
EC00339=-1108551,556475
EC00340=-1108551,556475
EC00341=-1108551,556475
EC00342=-1108551,556475
EC00343=-1108551,556475
EC00344=-1108551,556475
EC00345=-1108551,556475
EC00346=-1108551,556475
EC00347=-1108551,556475
EC00348=-1108551,556475
EC00349=-1108551,556475
EC00350=-1108551,556475
EC00351=-1108551,556475
EC00352=-1108551,556475
EC00353=-1108551,556475
EC00354=-1108551,556475
EC00355=-1108551,556475
EC00356=-1108551,556475
EC00357=-1108551,556475
EC00358=-1108551,556475
EC00359=-1108551,556475
EC00360=-1108551,556475
EC00361=-1108551,556475
EC00362=-1108551,556475
EC00363=-1108551,556475
EC00364=-1108551,556475
EC00365=-1108551,556475
EC00366=-1108551,556475
EC00367=-1108551,556475
EC00368=-1108551,556475
EC00369=-1108551,556475
EC00370=-1108551,556475
EC00371=-1108551,556475
EC00372=-1108551,556475
EC00373=-1108551,556475
EC00374=-1108551,556475
EC00375=-1108551,556475
EC00376=-1108551,556475
EC00377=-1108551,556475
EC00378=-1108551,556475
EC00379=-1108551,556475
EC00380=-1108551,556475
EC00381=-1108551,556475
EC00382=-1108551,556475
EC00383=-1108551,556475
EC00384=-1108551,556475
EC00385=-1108551,556475
EC00386=-1108551,556475
EC00387=-1108551,556475
EC00388=-1108551,556475
EC00389=-1108551,556475
EC00390=-1108551,556475
EC00391=-1108551,556475
EC00392=-1108551,556475
EC00393=-1108551,556475
EC00394=-1108551,556475
EC00395=-1108551,556475
EC00396=-1108551,556475
EC00397=-1108551,556475
EC00398=-1108551,556475
EC00399=-1108551,556475
EC00400=-1108551,556475
EC00401=-1108551,556475
EC00402=-1108551,556475
EC00403=-1108551,556475
EC00404=-1108551,556475
EC00405=-1108551,556475
EC00406=-1108551,556475
EC00407=-1108551,556475
EC00408=-1108551,556475
EC00409=-1108551,556475
EC00410=-1108551,556475
EC00411=-1108551,556475
EC00412=-1108551,556475
EC00413=-1108551,556475
EC00414=-1108551,556475
EC00415=-1108551,556475
EC00416=-1108551,556475
EC00417=-1108551,556475
EC00418=-1108551,556475
EC00419=-1108551,556475
EC00420=-1108551,556475
EC00421=-1108551,556475
EC00422=-1108551,556475
EC00423=-1108551,556475
EC00424=-1108551,556475
EC00425=-1108551,556475
EC00426=-1108551,556475
EC00427=-1108551,556475
EC00428=-1108551,556475
EC00429=-1108551,556475
EC00430=-1108551,556475
EC00431=-1108551,556475
EC00432=-1108551,556475
EC00433=-1108551,556475
EC00434=-1108551,556475
EC00435=-1108551,556475
EC00436=-1108551,556475
EC00437=-1108551,556475
EC00438=-1108551,556475
EC00439=-1108551,556475
EC00440=-1108551,556475
EC00441=-1108551,556475
EC00442=-1108551,556475
EC00443=-1108551,556475
EC00444=-1108551,556475
EC00445=-1108551,556475
EC00446=-1108551,556475
EC00447=-1108551,556475
EC00448=-1108551,556475
EC00449=-1108551,556475
EC00450=-1108551,556475
EC00451=-1108551,556475
EC00452=-1108551,556475
EC00453=-1108551,556475
EC00454=-1108551,556475
EC00455=-1108551,556475
EC00456=-1108551,556475
EC00457=-1108551,556475
EC00458=-1108551,556475
EC00459=-1108551,556475
EC00460=-1108551,556475
EC00461=-1108551,556475
EC00462=-1108551,556475
EC00463=-1108551,556475
EC00464=-1108551,556475
EC00465=-1108551,556475
EC00466=-1108551,556475
EC00467=-1108551,556475
EC00468=-1108551,556475
EC00469=-1108551,556475
EC00470=-1108551,556475
EC00471=-1108551,556475
EC00472=-1108551,556475
EC00473=-1108551,556475
EC00474=-1108551,556475
EC00475=-1108551,556475
EC00476=-1108551,556475
EC00477=-1108551,556475
EC00478=-1108551,556475
EC00479=-1108551,556475
EC00480=-1108551,556475
EC00481=-1108551,556475
EC00482=-1108551,556475
EC00483=-1108551,556475
EC00484=-1108551,556475
EC00485=-1108551,556475
EC00486=-1108551,556475
EC00487=-1108551,556475
EC00488=-1108551,556475
EC00489=-1108551,556475
EC00490=-1108551,556475
EC00491=-1108551,556475
EC00492=-1108551,556475
EC00493=-1108551,556475
EC00494=-1108551,556475
EC00495=-1108551,556475
EC00496=-1108551,556475
EC00497=-1108551,556475
EC00498=-1108551,556475
EC00499=-1108551,556475
EC00500=-1108551,556475
EC00501=-1108551,556475
EC00502=-1108551,556475
EC00503=-1108551,556475
EC00504=-1108551,556475
EC00505=-1108551,556475
EC00506=-1108551,556475
EC00507=-1108551,556475
EC00508=-1108551,556475
EC00509=-1108551,556475
EC00510=-1108551,556475
EC00511=-1108551,556475
EC00512=-1108551,556475
EC00513=-1108551,556475
EC00514=-1108551,556475
///POSTYPE BASE
///RECTAN
///RCONF 0,0,0,0,0,0,0,0,0,0,0,0,0,0,0,0,0,0,0,0,0,0,0,0
P00006=0.222,-3.123,-1.508,0.0000,0.0000,0.0000
P00021=-0.225,-6.128,-0.405,0.0000,0.0000,0.0000
P00022=0.222,-3.123,-1.508,0.0000,0.0000,0.0000
P00023=0.143,-0.036,0.682,0.0000,0.0000,0.0000
P00024=0.145,-0.552,1.326,0.0000,0.0000,0.0000
P00025=-2.003,0.006,0.728,0.0000,0.0000,0.0000
P00026=0.562,-0.002,-0.337,0.0000,0.0000,0.0000
P00027=-0.746,0.015,-9.096,0.0000,0.0000,0.0000
P00028=-2.237,-0.018,-7.702,0.0000,0.0000,0.0000
P00029=-2.156,-0.086,-4.681,0.0000,0.0000,0.0000
P00030=5.926,-4.294,-1.390,0.0000,0.0000,0.0000
P00031=1.853,-0.001,-1.549,0.0000,0.0000,0.0000
P00032=1.957,0.503,-7.217,0.0000,0.0000,0.0000
///RCONF 0,0,0,0,1,0,0,0,0,0,0,0,0,0,0,0,0,0,0,0,0,0,0,0
P00033=-0.123,0.612,-5.012,0.0000,0.0000,0.0000
///RCONF 0,0,0,0,0,0,0,0,0,0,0,0,0,0,0,0,0,0,0,0,0,0,0,0
P00041=0.192,3.924,0.305,0.0000,0.0000,0.0000
P00042=-0.217,1.941,0.413,0.0000,0.0000,0.0000
P00043=-0.044,-1.937,1.197,0.0000,0.0000,0.0000
P00044=0.687,-2.322,1.156,0.0000,0.0000,0.0000
P00045=-0.068,-0.810,1.603,0.0000,0.0000,0.0000
P00046=0.799,0.043,1.292,0.0000,0.0000,0.0000
///RCONF 0,1,0,0,0,0,0,0,0,0,0,0,0,0,0,0,0,0,0,0,0,0,0,0
P00047=-0.011,1.737,-0.646,0.0000,0.0000,0.0000
///RCONF 0,0,0,0,0,0,0,0,0,0,0,0,0,0,0,0,0,0,0,0,0,0,0,0
P00048=2.411,0.025,-0.606,0.0000,0.0000,0.0000
P00049=3.413,-3.572,-1.618,0.0000,0.0000,0.0000
P00050=4.296,-4.501,-0.826,0.0000,0.0000,0.0000
P00051=0.367,3.892,0.009,0.0000,0.0000,0.0000
P00052=0.088,2.832,-0.342,0.0000,0.0000,0.0000
P00053=0.134,6.594,0.107,0.0000,0.0000,0.0000
//INST
///DATE 2024/02/02 10:05
///ATTR SC,RW
///GROUP1 RB1,BS1
///GROUP2 ST1
NOP
'N_r2_D100(P)(125,-90)
'
MOVJ C00000 BC00000 VJ=100.00  +MOVJ EC00000 VJ=100.00
MOVJ C00001 BC00001 VJ=100.00  +MOVJ EC00001 VJ=100.00
'
MOVJ C00002 BC00002 VJ=100.00  +MOVJ EC00002 VJ=100.00
MOVJ C00003 BC00003 VJ=100.00  +MOVJ EC00003 VJ=100.00
MOVJ C00004 BC00004 VJ=100.00  +MOVJ EC00004 VJ=100.00
MOVJ C00005 BC00005 VJ=100.00  +MOVJ EC00005 VJ=100.00
MOVJ C00006 BC00006 VJ=100.00  +MOVJ EC00006 VJ=100.00
'Path S3336
SSFTOF
MOVJ C00007 BC00007 VJ=100.00  +MOVJ EC00007 VJ=100.00
MOVL C00008 BC00008 V=400.0  +MOVJ EC00008 VJ=100.00
SMOVL C00009 BC00009 V=100.0  +MOVJ EC00009
SREFP 3 C00010 BC00010  +REFP EC00010
CALL JOB:SEARCH-R1-S1
SET P021 P006
SSFTON P021
SMOVL C00011 BC00011 V=100.0  +MOVJ EC00011
SMOVL C00012 BC00012 V=100.0  +MOVJ EC00012
SREFP 3 C00013 BC00013  +REFP EC00013
CALL JOB:SEARCH-R1-S1
SET P021 P006
SSFTON P021
SMOVL C00014 BC00014 V=100.0  +MOVJ EC00014
MOVL C00015 BC00015 V=400.0  +MOVJ EC00015 VJ=100.00
MOVL C00016 BC00016 V=1000.0  +MOVJ EC00016 VJ=100.00
'Path S3337
SSFTOF
MOVJ C00017 BC00017 VJ=100.00  +MOVJ EC00017 VJ=100.00
MOVL C00018 BC00018 V=400.0  +MOVJ EC00018 VJ=100.00
SMOVL C00019 BC00019 V=100.0  +MOVJ EC00019
SREFP 3 C00020 BC00020  +REFP EC00020
CALL JOB:SEARCH-R1-S1
SET P022 P006
SSFTON P022
SMOVL C00021 BC00021 V=100.0  +MOVJ EC00021
SMOVL C00022 BC00022 V=100.0  +MOVJ EC00022
SREFP 3 C00023 BC00023  +REFP EC00023
CALL JOB:SEARCH-R1-S1
SET P022 P006
SSFTON P022
SMOVL C00024 BC00024 V=100.0  +MOVJ EC00024
MOVL C00025 BC00025 V=400.0  +MOVJ EC00025 VJ=100.00
MOVL C00026 BC00026 V=1000.0  +MOVJ EC00026 VJ=100.00
'Path S3338
SSFTOF
MOVJ C00027 BC00027 VJ=100.00  +MOVJ EC00027 VJ=100.00
MOVL C00028 BC00028 V=400.0  +MOVJ EC00028 VJ=100.00
SMOVL C00029 BC00029 V=100.0  +MOVJ EC00029
SREFP 3 C00030 BC00030  +REFP EC00030
CALL JOB:SEARCH-R1-S1
SET P023 P006
SSFTON P023
SMOVL C00031 BC00031 V=100.0  +MOVJ EC00031
SMOVL C00032 BC00032 V=100.0  +MOVJ EC00032
SREFP 3 C00033 BC00033  +REFP EC00033
CALL JOB:SEARCH-R1-S1
SET P023 P006
SSFTON P023
SMOVL C00034 BC00034 V=100.0  +MOVJ EC00034
MOVL C00035 BC00035 V=400.0  +MOVJ EC00035 VJ=100.00
MOVL C00036 BC00036 V=1000.0  +MOVJ EC00036 VJ=100.00
MOVJ C00037 BC00037 VJ=100.00  +MOVJ EC00037 VJ=100.00
'Path S3339
SSFTOF
MOVJ C00038 BC00038 VJ=100.00  +MOVJ EC00038 VJ=100.00
MOVL C00039 BC00039 V=400.0  +MOVJ EC00039 VJ=100.00
SMOVL C00040 BC00040 V=100.0  +MOVJ EC00040
SREFP 3 C00041 BC00041  +REFP EC00041
CALL JOB:SEARCH-R1-S1
SET P024 P006
SSFTON P024
SMOVL C00042 BC00042 V=100.0  +MOVJ EC00042
SMOVL C00043 BC00043 V=100.0  +MOVJ EC00043
SREFP 3 C00044 BC00044  +REFP EC00044
CALL JOB:SEARCH-R1-S1
SET P024 P006
SSFTON P024
SMOVL C00045 BC00045 V=100.0  +MOVJ EC00045
MOVL C00046 BC00046 V=400.0  +MOVJ EC00046 VJ=100.00
MOVL C00047 BC00047 V=1000.0  +MOVJ EC00047 VJ=100.00
'Path S3341
SSFTOF
MOVJ C00048 BC00048 VJ=100.00  +MOVJ EC00048 VJ=100.00
MOVL C00049 BC00049 V=400.0  +MOVJ EC00049 VJ=100.00
SMOVL C00050 BC00050 V=100.0  +MOVJ EC00050
SREFP 3 C00051 BC00051  +REFP EC00051
CALL JOB:SEARCH-R1-S1
SET P025 P006
SSFTON P025
SMOVL C00052 BC00052 V=100.0  +MOVJ EC00052
SMOVL C00053 BC00053 V=100.0  +MOVJ EC00053
SREFP 3 C00054 BC00054  +REFP EC00054
CALL JOB:SEARCH-R1-S1
SET P025 P006
SSFTON P025
SMOVL C00055 BC00055 V=100.0  +MOVJ EC00055
MOVL C00056 BC00056 V=400.0  +MOVJ EC00056 VJ=100.00
MOVL C00057 BC00057 V=1000.0  +MOVJ EC00057 VJ=100.00
'Path S3343
SSFTOF
MOVJ C00058 BC00058 VJ=100.00  +MOVJ EC00058 VJ=100.00
MOVL C00059 BC00059 V=400.0  +MOVJ EC00059 VJ=100.00
SMOVL C00060 BC00060 V=100.0  +MOVJ EC00060
SREFP 3 C00061 BC00061  +REFP EC00061
CALL JOB:SEARCH-R1-S1
SET P026 P006
SSFTON P026
SMOVL C00062 BC00062 V=100.0  +MOVJ EC00062
SMOVL C00063 BC00063 V=100.0  +MOVJ EC00063
SREFP 3 C00064 BC00064  +REFP EC00064
CALL JOB:SEARCH-R1-S1
SET P026 P006
SSFTON P026
SMOVL C00065 BC00065 V=100.0  +MOVJ EC00065
MOVL C00066 BC00066 V=400.0  +MOVJ EC00066 VJ=100.00
MOVL C00067 BC00067 V=1000.0  +MOVJ EC00067 VJ=100.00
MOVJ C00068 BC00068 VJ=100.00  +MOVJ EC00068 VJ=100.00
'Path S3345
SSFTOF
MOVJ C00069 BC00069 VJ=100.00  +MOVJ EC00069 VJ=100.00
MOVL C00070 BC00070 V=400.0  +MOVJ EC00070 VJ=100.00
SMOVL C00071 BC00071 V=100.0  +MOVJ EC00071
SREFP 3 C00072 BC00072  +REFP EC00072
CALL JOB:SEARCH-R1-S1
SET P027 P006
SSFTON P027
SMOVL C00073 BC00073 V=100.0  +MOVJ EC00073
SMOVL C00074 BC00074 V=100.0  +MOVJ EC00074
SREFP 3 C00075 BC00075  +REFP EC00075
CALL JOB:SEARCH-R1-S1
SET P027 P006
SSFTON P027
SMOVL C00076 BC00076 V=100.0  +MOVJ EC00076
MOVL C00077 BC00077 V=400.0  +MOVJ EC00077 VJ=100.00
MOVL C00078 BC00078 V=1000.0  +MOVJ EC00078 VJ=100.00
MOVJ C00079 BC00079 VJ=100.00  +MOVJ EC00079 VJ=100.00
'Path S3347
SSFTOF
MOVJ C00080 BC00080 VJ=100.00  +MOVJ EC00080 VJ=100.00
MOVL C00081 BC00081 V=400.0  +MOVJ EC00081 VJ=100.00
SMOVL C00082 BC00082 V=100.0  +MOVJ EC00082
SREFP 3 C00083 BC00083  +REFP EC00083
CALL JOB:SEARCH-R1-S1
SET P028 P006
SSFTON P028
SMOVL C00084 BC00084 V=100.0  +MOVJ EC00084
SMOVL C00085 BC00085 V=100.0  +MOVJ EC00085
SREFP 3 C00086 BC00086  +REFP EC00086
CALL JOB:SEARCH-R1-S1
SET P028 P006
SSFTON P028
SMOVL C00087 BC00087 V=100.0  +MOVJ EC00087
MOVL C00088 BC00088 V=400.0  +MOVJ EC00088 VJ=100.00
MOVL C00089 BC00089 V=1000.0  +MOVJ EC00089 VJ=100.00
'Path S3349
SSFTOF
MOVJ C00090 BC00090 VJ=100.00  +MOVJ EC00090 VJ=100.00
MOVL C00091 BC00091 V=400.0  +MOVJ EC00091 VJ=100.00
SMOVL C00092 BC00092 V=100.0  +MOVJ EC00092
SREFP 3 C00093 BC00093  +REFP EC00093
CALL JOB:SEARCH-R1-S1
SET P029 P006
SSFTON P029
SMOVL C00094 BC00094 V=100.0  +MOVJ EC00094
SMOVL C00095 BC00095 V=100.0  +MOVJ EC00095
SREFP 3 C00096 BC00096  +REFP EC00096
CALL JOB:SEARCH-R1-S1
SET P029 P006
SSFTON P029
SMOVL C00097 BC00097 V=100.0  +MOVJ EC00097
MOVL C00098 BC00098 V=400.0  +MOVJ EC00098 VJ=100.00
MOVL C00099 BC00099 V=1000.0  +MOVJ EC00099 VJ=100.00
'Path S3350
SSFTOF
MOVJ C00100 BC00100 VJ=100.00  +MOVJ EC00100 VJ=100.00
MOVL C00101 BC00101 V=400.0  +MOVJ EC00101 VJ=100.00
SMOVL C00102 BC00102 V=100.0  +MOVJ EC00102
SREFP 3 C00103 BC00103  +REFP EC00103
CALL JOB:SEARCH-R1-S1
SET P030 P006
SSFTON P030
SMOVL C00104 BC00104 V=100.0  +MOVJ EC00104
SMOVL C00105 BC00105 V=100.0  +MOVJ EC00105
SREFP 3 C00106 BC00106  +REFP EC00106
CALL JOB:SEARCH-R1-S1
SET P030 P006
SSFTON P030
SMOVL C00107 BC00107 V=100.0  +MOVJ EC00107
SMOVL C00108 BC00108 V=100.0  +MOVJ EC00108
SREFP 3 C00109 BC00109  +REFP EC00109
CALL JOB:SEARCH-R1-S1
SET P030 P006
SSFTON P030
SMOVL C00110 BC00110 V=100.0  +MOVJ EC00110
MOVL C00111 BC00111 V=400.0  +MOVJ EC00111 VJ=100.00
MOVL C00112 BC00112 V=1000.0  +MOVJ EC00112 VJ=100.00
'Path S3351
SSFTOF
MOVJ C00113 BC00113 VJ=100.00  +MOVJ EC00113 VJ=100.00
MOVL C00114 BC00114 V=400.0  +MOVJ EC00114 VJ=100.00
SMOVL C00115 BC00115 V=100.0  +MOVJ EC00115
SREFP 3 C00116 BC00116  +REFP EC00116
CALL JOB:SEARCH-R1-S1
SET P031 P006
SSFTON P031
SMOVL C00117 BC00117 V=100.0  +MOVJ EC00117
SMOVL C00118 BC00118 V=100.0  +MOVJ EC00118
SREFP 3 C00119 BC00119  +REFP EC00119
CALL JOB:SEARCH-R1-S1
SET P031 P006
SSFTON P031
SMOVL C00120 BC00120 V=100.0  +MOVJ EC00120
MOVL C00121 BC00121 V=400.0  +MOVJ EC00121 VJ=100.00
MOVL C00122 BC00122 V=1000.0  +MOVJ EC00122 VJ=100.00
MOVJ C00123 BC00123 VJ=100.00  +MOVJ EC00123 VJ=100.00
'Path S3352
SSFTOF
MOVJ C00124 BC00124 VJ=100.00  +MOVJ EC00124 VJ=100.00
MOVL C00125 BC00125 V=400.0  +MOVJ EC00125 VJ=100.00
SMOVL C00126 BC00126 V=100.0  +MOVJ EC00126
SREFP 3 C00127 BC00127  +REFP EC00127
CALL JOB:SEARCH-R1-S1
SET P032 P006
SSFTON P032
SMOVL C00128 BC00128 V=100.0  +MOVJ EC00128
SMOVL C00129 BC00129 V=100.0  +MOVJ EC00129
SREFP 3 C00130 BC00130  +REFP EC00130
CALL JOB:SEARCH-R1-S1
SET P032 P006
SSFTON P032
SMOVL C00131 BC00131 V=100.0  +MOVJ EC00131
MOVL C00132 BC00132 V=400.0  +MOVJ EC00132 VJ=100.00
MOVL C00133 BC00133 V=1000.0  +MOVJ EC00133 VJ=100.00
'Path S3353
SSFTOF
MOVJ C00134 BC00134 VJ=100.00  +MOVJ EC00134 VJ=100.00
MOVL C00135 BC00135 V=400.0  +MOVJ EC00135 VJ=100.00
SMOVL C00136 BC00136 V=100.0  +MOVJ EC00136
SREFP 3 C00137 BC00137  +REFP EC00137
CALL JOB:SEARCH-R1-S1
SET P033 P006
SSFTON P033
SMOVL C00138 BC00138 V=100.0  +MOVJ EC00138
SMOVL C00139 BC00139 V=100.0  +MOVJ EC00139
SREFP 3 C00140 BC00140  +REFP EC00140
CALL JOB:SEARCH-R1-S1
SET P033 P006
SSFTON P033
SMOVL C00141 BC00141 V=100.0  +MOVJ EC00141
MOVL C00142 BC00142 V=400.0  +MOVJ EC00142 VJ=100.00
MOVL C00143 BC00143 V=1000.0  +MOVJ EC00143 VJ=100.00
MOVJ C00144 BC00144 VJ=100.00  +MOVJ EC00144 VJ=100.00
MOVJ C00145 BC00145 VJ=100.00  +MOVJ EC00145 VJ=100.00
'Path W3292
SSFTOF
SSFTON P021
MOVJ C00146 BC00146 VJ=100.00  +MOVJ EC00146 VJ=100.00
SMOVL C00147 BC00147 V=400.0  +MOVJ EC00147
SMOVL C00148 BC00148 V=100.0 PL=0  +MOVJ EC00148
SREFP 1 C00149 BC00149  +REFP EC00149
SREFP 2 C00150 BC00150  +REFP EC00150
MACRO1 MJ#(0) ARGF0
ARCON
SMOVL C00151 BC00151 V=10.0  +MOVJ EC00151
SMOVL C00152 BC00152 V=10.0  +MOVJ EC00152
SMOVL C00153 BC00153 V=10.0  +MOVJ EC00153
ARCOF
SMOVL C00154 BC00154 V=400.0  +MOVJ EC00154
SMOVL C00155 BC00155 V=1000.0  +MOVJ EC00155
SSFTOF
'Path W3293
SSFTOF
SSFTON P022
MOVJ C00156 BC00156 VJ=100.00  +MOVJ EC00156 VJ=100.00
SMOVL C00157 BC00157 V=400.0  +MOVJ EC00157
SMOVL C00158 BC00158 V=100.0 PL=0  +MOVJ EC00158
SREFP 1 C00159 BC00159  +REFP EC00159
SREFP 2 C00160 BC00160  +REFP EC00160
MACRO1 MJ#(0) ARGF0
ARCON
SMOVL C00161 BC00161 V=10.0  +MOVJ EC00161
SMOVL C00162 BC00162 V=10.0  +MOVJ EC00162
SMOVL C00163 BC00163 V=10.0  +MOVJ EC00163
ARCOF
SMOVL C00164 BC00164 V=400.0  +MOVJ EC00164
SMOVL C00165 BC00165 V=1000.0  +MOVJ EC00165
SSFTOF
'Path W3294
SSFTOF
SSFTON P023
MOVJ C00166 BC00166 VJ=100.00  +MOVJ EC00166 VJ=100.00
SMOVL C00167 BC00167 V=400.0  +MOVJ EC00167
SMOVL C00168 BC00168 V=100.0 PL=0  +MOVJ EC00168
SREFP 1 C00169 BC00169  +REFP EC00169
SREFP 2 C00170 BC00170  +REFP EC00170
MACRO1 MJ#(0) ARGF0
ARCON
SMOVL C00171 BC00171 V=10.0  +MOVJ EC00171
SMOVL C00172 BC00172 V=10.0  +MOVJ EC00172
SMOVL C00173 BC00173 V=10.0  +MOVJ EC00173
ARCOF
SMOVL C00174 BC00174 V=400.0  +MOVJ EC00174
SMOVL C00175 BC00175 V=1000.0  +MOVJ EC00175
SSFTOF
'
MOVJ C00176 BC00176 VJ=100.00  +MOVJ EC00176 VJ=100.00
'Path W3340
SSFTOF
SSFTON P024
MOVJ C00177 BC00177 VJ=100.00  +MOVJ EC00177 VJ=100.00
SMOVL C00178 BC00178 V=400.0  +MOVJ EC00178
SMOVL C00179 BC00179 V=150.0 PL=0  +MOVJ EC00179
SREFP 1 C00180 BC00180  +REFP EC00180
SREFP 2 C00181 BC00181  +REFP EC00181
MACRO1 MJ#(0) ARGF0
ARCON
SMOVL C00182 BC00182 V=10.0  +MOVJ EC00182
SMOVL C00183 BC00183 V=10.0  +MOVJ EC00183
SMOVL C00184 BC00184 V=10.0  +MOVJ EC00184
ARCOF
SMOVL C00185 BC00185 V=400.0  +MOVJ EC00185
SMOVL C00186 BC00186 V=1000.0  +MOVJ EC00186
SSFTOF
'Path W3342
SSFTOF
SSFTON P025
MOVJ C00187 BC00187 VJ=100.00  +MOVJ EC00187 VJ=100.00
SMOVL C00188 BC00188 V=400.0  +MOVJ EC00188
SMOVL C00189 BC00189 V=150.0 PL=0  +MOVJ EC00189
SREFP 1 C00190 BC00190  +REFP EC00190
SREFP 2 C00191 BC00191  +REFP EC00191
MACRO1 MJ#(0) ARGF0
ARCON
SMOVL C00192 BC00192 V=10.0  +MOVJ EC00192
SMOVL C00193 BC00193 V=10.0  +MOVJ EC00193
SMOVL C00194 BC00194 V=10.0  +MOVJ EC00194
ARCOF
SMOVL C00195 BC00195 V=400.0  +MOVJ EC00195
SMOVL C00196 BC00196 V=1000.0  +MOVJ EC00196
SSFTOF
'Path W3344
SSFTOF
SSFTON P026
MOVJ C00197 BC00197 VJ=100.00  +MOVJ EC00197 VJ=100.00
SMOVL C00198 BC00198 V=400.0  +MOVJ EC00198
SMOVL C00199 BC00199 V=150.0 PL=0  +MOVJ EC00199
SREFP 1 C00200 BC00200  +REFP EC00200
SREFP 2 C00201 BC00201  +REFP EC00201
MACRO1 MJ#(0) ARGF0
ARCON
SMOVL C00202 BC00202 V=10.0  +MOVJ EC00202
SMOVL C00203 BC00203 V=10.0  +MOVJ EC00203
SMOVL C00204 BC00204 V=10.0  +MOVJ EC00204
ARCOF
SMOVL C00205 BC00205 V=400.0  +MOVJ EC00205
SMOVL C00206 BC00206 V=1000.0  +MOVJ EC00206
SSFTOF
'
MOVJ C00207 BC00207 VJ=100.00  +MOVJ EC00207 VJ=100.00
'Path W3346
SSFTOF
SSFTON P027
MOVJ C00208 BC00208 VJ=100.00  +MOVJ EC00208 VJ=100.00
SMOVL C00209 BC00209 V=400.0  +MOVJ EC00209
SMOVL C00210 BC00210 V=150.0 PL=0  +MOVJ EC00210
SREFP 1 C00211 BC00211  +REFP EC00211
SREFP 2 C00212 BC00212  +REFP EC00212
MACRO1 MJ#(0) ARGF0
ARCON
SMOVL C00213 BC00213 V=10.0  +MOVJ EC00213
SMOVL C00214 BC00214 V=10.0  +MOVJ EC00214
SMOVL C00215 BC00215 V=10.0  +MOVJ EC00215
ARCOF
SMOVL C00216 BC00216 V=400.0  +MOVJ EC00216
SMOVL C00217 BC00217 V=1000.0  +MOVJ EC00217
SSFTOF
'Path W3348
SSFTOF
SSFTON P028
MOVJ C00218 BC00218 VJ=100.00  +MOVJ EC00218 VJ=100.00
SMOVL C00219 BC00219 V=400.0  +MOVJ EC00219
SMOVL C00220 BC00220 V=150.0 PL=0  +MOVJ EC00220
SREFP 1 C00221 BC00221  +REFP EC00221
SREFP 2 C00222 BC00222  +REFP EC00222
MACRO1 MJ#(0) ARGF0
ARCON
SMOVL C00223 BC00223 V=10.0  +MOVJ EC00223
SMOVL C00224 BC00224 V=10.0  +MOVJ EC00224
SMOVL C00225 BC00225 V=10.0  +MOVJ EC00225
ARCOF
SMOVL C00226 BC00226 V=400.0  +MOVJ EC00226
SMOVL C00227 BC00227 V=1000.0  +MOVJ EC00227
SSFTOF
'Path W3350
SSFTOF
SSFTON P029
MOVJ C00228 BC00228 VJ=100.00  +MOVJ EC00228 VJ=100.00
SMOVL C00229 BC00229 V=400.0  +MOVJ EC00229
SMOVL C00230 BC00230 V=150.0 PL=0  +MOVJ EC00230
SREFP 1 C00231 BC00231  +REFP EC00231
SREFP 2 C00232 BC00232  +REFP EC00232
MACRO1 MJ#(0) ARGF0
ARCON
SMOVL C00233 BC00233 V=10.0  +MOVJ EC00233
SMOVL C00234 BC00234 V=10.0  +MOVJ EC00234
SMOVL C00235 BC00235 V=10.0  +MOVJ EC00235
ARCOF
SMOVL C00236 BC00236 V=400.0  +MOVJ EC00236
SMOVL C00237 BC00237 V=1000.0  +MOVJ EC00237
SSFTOF
MOVJ C00238 BC00238 VJ=100.00  +MOVJ EC00238 VJ=100.00
'
'Path W3316
SSFTOF
SSFTON P031
MOVJ C00239 BC00239 VJ=100.00  +MOVJ EC00239 VJ=100.00
SMOVL C00240 BC00240 V=400.0  +MOVJ EC00240
SMOVL C00241 BC00241 V=150.0 PL=0  +MOVJ EC00241
SREFP 1 C00242 BC00242  +REFP EC00242
SREFP 2 C00243 BC00243  +REFP EC00243
MACRO1 MJ#(0) ARGF0
ARCON
SMOVL C00244 BC00244 V=10.0  +MOVJ EC00244
SSFTON P030
SMOVL C00245 BC00245 V=10.0  +MOVJ EC00245
SMOVL C00246 BC00246 V=10.0  +MOVJ EC00246
ARCOF
SMOVL C00247 BC00247 V=400.0  +MOVJ EC00247
SMOVL C00248 BC00248 V=1000.0  +MOVJ EC00248
SSFTOF
MOVJ C00249 BC00249 VJ=100.00  +MOVJ EC00249 VJ=100.00
'
'Path W3319
SSFTOF
SSFTON P032
MOVJ C00250 BC00250 VJ=100.00  +MOVJ EC00250 VJ=100.00
SMOVL C00251 BC00251 V=400.0  +MOVJ EC00251
SMOVL C00252 BC00252 V=150.0 PL=0  +MOVJ EC00252
SREFP 1 C00253 BC00253  +REFP EC00253
SREFP 2 C00254 BC00254  +REFP EC00254
MACRO1 MJ#(0) ARGF0
ARCON
SSFTON P033
SMOVL C00255 BC00255 V=10.0  +MOVJ EC00255
ARCOF
SMOVL C00256 BC00256 V=400.0  +MOVJ EC00256
SMOVL C00257 BC00257 V=1000.0  +MOVJ EC00257
SSFTOF
MOVJ C00258 BC00258 VJ=100.00  +MOVJ EC00258 VJ=100.00
MOVJ C00259 BC00259 VJ=100.00  +MOVJ EC00259 VJ=100.00
'
MOVJ C00260 BC00260 VJ=100.00  +MOVJ EC00260 VJ=100.00
MOVJ C00261 BC00261 VJ=100.00  +MOVJ EC00261 VJ=100.00
'CUT-WIRE !!!!
MOVJ C00262 BC00262 VJ=100.00  +MOVJ EC00262 VJ=100.00
MOVJ C00263 BC00263 VJ=100.00  +MOVJ EC00263 VJ=100.00
MOVJ C00264 BC00264 VJ=100.00  +MOVJ EC00264 VJ=100.00
MOVJ C00265 BC00265 VJ=100.00  +MOVJ EC00265 VJ=100.00
'
'Path S3355
SSFTOF
MOVJ C00266 BC00266 VJ=100.00  +MOVJ EC00266 VJ=100.00
MOVL C00267 BC00267 V=400.0  +MOVJ EC00267 VJ=100.00
SMOVL C00268 BC00268 V=100.0  +MOVJ EC00268
SREFP 3 C00269 BC00269  +REFP EC00269
CALL JOB:SEARCH-R1-S1
SET P041 P006
SSFTON P041
SMOVL C00270 BC00270 V=100.0  +MOVJ EC00270
SMOVL C00271 BC00271 V=100.0  +MOVJ EC00271
SREFP 3 C00272 BC00272  +REFP EC00272
CALL JOB:SEARCH-R1-S1
SET P041 P006
SSFTON P041
SMOVL C00273 BC00273 V=100.0  +MOVJ EC00273
MOVL C00274 BC00274 V=400.0  +MOVJ EC00274 VJ=100.00
MOVL C00275 BC00275 V=1000.0  +MOVJ EC00275 VJ=100.00
'Path S3356
SSFTOF
MOVJ C00276 BC00276 VJ=100.00  +MOVJ EC00276 VJ=100.00
MOVL C00277 BC00277 V=400.0  +MOVJ EC00277 VJ=100.00
SMOVL C00278 BC00278 V=100.0  +MOVJ EC00278
SREFP 3 C00279 BC00279  +REFP EC00279
CALL JOB:SEARCH-R1-S1
SET P042 P006
SSFTON P042
SMOVL C00280 BC00280 V=100.0  +MOVJ EC00280
SMOVL C00281 BC00281 V=100.0  +MOVJ EC00281
SREFP 3 C00282 BC00282  +REFP EC00282
CALL JOB:SEARCH-R1-S1
SET P042 P006
SSFTON P042
SMOVL C00283 BC00283 V=100.0  +MOVJ EC00283
MOVL C00284 BC00284 V=400.0  +MOVJ EC00284 VJ=100.00
MOVL C00285 BC00285 V=1000.0  +MOVJ EC00285 VJ=100.00
MOVJ C00286 BC00286 VJ=100.00  +MOVJ EC00286 VJ=100.00
'Path S3357
SSFTOF
MOVJ C00287 BC00287 VJ=100.00  +MOVJ EC00287 VJ=100.00
MOVL C00288 BC00288 V=400.0  +MOVJ EC00288 VJ=100.00
SMOVL C00289 BC00289 V=100.0  +MOVJ EC00289
SREFP 3 C00290 BC00290  +REFP EC00290
CALL JOB:SEARCH-R1-S1
SET P043 P006
SSFTON P043
SMOVL C00291 BC00291 V=100.0  +MOVJ EC00291
SMOVL C00292 BC00292 V=100.0  +MOVJ EC00292
SREFP 3 C00293 BC00293  +REFP EC00293
CALL JOB:SEARCH-R1-S1
SET P043 P006
SSFTON P043
SMOVL C00294 BC00294 V=100.0  +MOVJ EC00294
MOVL C00295 BC00295 V=400.0  +MOVJ EC00295 VJ=100.00
MOVL C00296 BC00296 V=1000.0  +MOVJ EC00296 VJ=100.00
MOVJ C00297 BC00297 VJ=100.00  +MOVJ EC00297 VJ=100.00
'Path S3358
SSFTOF
MOVJ C00298 BC00298 VJ=100.00  +MOVJ EC00298 VJ=100.00
MOVL C00299 BC00299 V=400.0  +MOVJ EC00299 VJ=100.00
SMOVL C00300 BC00300 V=100.0  +MOVJ EC00300
SREFP 3 C00301 BC00301  +REFP EC00301
CALL JOB:SEARCH-R1-S1
SET P044 P006
SSFTON P044
SMOVL C00302 BC00302 V=100.0  +MOVJ EC00302
SMOVL C00303 BC00303 V=100.0  +MOVJ EC00303
SREFP 3 C00304 BC00304  +REFP EC00304
CALL JOB:SEARCH-R1-S1
SET P044 P006
SSFTON P044
SMOVL C00305 BC00305 V=100.0  +MOVJ EC00305
MOVL C00306 BC00306 V=400.0  +MOVJ EC00306 VJ=100.00
MOVL C00307 BC00307 V=1000.0  +MOVJ EC00307 VJ=100.00
'Path S3359
SSFTOF
MOVJ C00308 BC00308 VJ=100.00  +MOVJ EC00308 VJ=100.00
MOVL C00309 BC00309 V=400.0  +MOVJ EC00309 VJ=100.00
SMOVL C00310 BC00310 V=100.0  +MOVJ EC00310
SREFP 3 C00311 BC00311  +REFP EC00311
CALL JOB:SEARCH-R1-S1
SET P045 P006
SSFTON P045
SMOVL C00312 BC00312 V=100.0  +MOVJ EC00312
SMOVL C00313 BC00313 V=100.0  +MOVJ EC00313
SREFP 3 C00314 BC00314  +REFP EC00314
CALL JOB:SEARCH-R1-S1
SET P045 P006
SSFTON P045
SMOVL C00315 BC00315 V=100.0  +MOVJ EC00315
MOVL C00316 BC00316 V=400.0  +MOVJ EC00316 VJ=100.00
MOVL C00317 BC00317 V=1000.0  +MOVJ EC00317 VJ=100.00
'Path S3360
SSFTOF
MOVJ C00318 BC00318 VJ=100.00  +MOVJ EC00318 VJ=100.00
MOVL C00319 BC00319 V=400.0  +MOVJ EC00319 VJ=100.00
SMOVL C00320 BC00320 V=100.0  +MOVJ EC00320
SREFP 3 C00321 BC00321  +REFP EC00321
CALL JOB:SEARCH-R1-S1
SET P046 P006
SSFTON P046
SMOVL C00322 BC00322 V=100.0  +MOVJ EC00322
SMOVL C00323 BC00323 V=100.0  +MOVJ EC00323
SREFP 3 C00324 BC00324  +REFP EC00324
CALL JOB:SEARCH-R1-S1
SET P046 P006
SSFTON P046
SMOVL C00325 BC00325 V=100.0  +MOVJ EC00325
MOVL C00326 BC00326 V=400.0  +MOVJ EC00326 VJ=100.00
MOVL C00327 BC00327 V=1000.0  +MOVJ EC00327 VJ=100.00
MOVJ C00328 BC00328 VJ=100.00  +MOVJ EC00328 VJ=100.00
'Path S3361
SSFTOF
MOVJ C00329 BC00329 VJ=100.00  +MOVJ EC00329 VJ=100.00
MOVL C00330 BC00330 V=400.0  +MOVJ EC00330 VJ=100.00
SMOVL C00331 BC00331 V=100.0  +MOVJ EC00331
SREFP 3 C00332 BC00332  +REFP EC00332
CALL JOB:SEARCH-R1-S1
SET P047 P006
SSFTON P047
SMOVL C00333 BC00333 V=100.0  +MOVJ EC00333
SMOVL C00334 BC00334 V=100.0  +MOVJ EC00334
SREFP 3 C00335 BC00335  +REFP EC00335
CALL JOB:SEARCH-R1-S1
SET P047 P006
SSFTON P047
SMOVL C00336 BC00336 V=100.0  +MOVJ EC00336
MOVL C00337 BC00337 V=400.0  +MOVJ EC00337 VJ=100.00
MOVL C00338 BC00338 V=1000.0  +MOVJ EC00338 VJ=100.00
'Path S3362
SSFTOF
MOVJ C00339 BC00339 VJ=100.00  +MOVJ EC00339 VJ=100.00
MOVL C00340 BC00340 V=400.0  +MOVJ EC00340 VJ=100.00
SMOVL C00341 BC00341 V=100.0  +MOVJ EC00341
SREFP 3 C00342 BC00342  +REFP EC00342
CALL JOB:SEARCH-R1-S1
SET P048 P006
SSFTON P048
SMOVL C00343 BC00343 V=100.0  +MOVJ EC00343
SMOVL C00344 BC00344 V=100.0  +MOVJ EC00344
SREFP 3 C00345 BC00345  +REFP EC00345
CALL JOB:SEARCH-R1-S1
SET P048 P006
SSFTON P048
SMOVL C00346 BC00346 V=100.0  +MOVJ EC00346
MOVL C00347 BC00347 V=400.0  +MOVJ EC00347 VJ=100.00
MOVL C00348 BC00348 V=1000.0  +MOVJ EC00348 VJ=100.00
'Path S3363
SSFTOF
MOVJ C00349 BC00349 VJ=100.00  +MOVJ EC00349 VJ=100.00
MOVL C00350 BC00350 V=400.0  +MOVJ EC00350 VJ=100.00
SMOVL C00351 BC00351 V=100.0  +MOVJ EC00351
SREFP 3 C00352 BC00352  +REFP EC00352
CALL JOB:SEARCH-R1-S1
SET P049 P006
SSFTON P049
SMOVL C00353 BC00353 V=100.0  +MOVJ EC00353
SMOVL C00354 BC00354 V=100.0  +MOVJ EC00354
SREFP 3 C00355 BC00355  +REFP EC00355
CALL JOB:SEARCH-R1-S1
SET P049 P006
SSFTON P049
SMOVL C00356 BC00356 V=100.0  +MOVJ EC00356
MOVL C00357 BC00357 V=400.0  +MOVJ EC00357 VJ=100.00
MOVL C00358 BC00358 V=1000.0  +MOVJ EC00358 VJ=100.00
'Path S3364
SSFTOF
MOVJ C00359 BC00359 VJ=100.00  +MOVJ EC00359 VJ=100.00
MOVL C00360 BC00360 V=400.0  +MOVJ EC00360 VJ=100.00
SMOVL C00361 BC00361 V=100.0  +MOVJ EC00361
SREFP 3 C00362 BC00362  +REFP EC00362
CALL JOB:SEARCH-R1-S1
SET P050 P006
SSFTON P050
SMOVL C00363 BC00363 V=100.0  +MOVJ EC00363
SMOVL C00364 BC00364 V=100.0  +MOVJ EC00364
SREFP 3 C00365 BC00365  +REFP EC00365
CALL JOB:SEARCH-R1-S1
SET P050 P006
SSFTON P050
SMOVL C00366 BC00366 V=100.0  +MOVJ EC00366
SMOVL C00367 BC00367 V=100.0  +MOVJ EC00367
SREFP 3 C00368 BC00368  +REFP EC00368
CALL JOB:SEARCH-R1-S1
SET P050 P006
SSFTON P050
SMOVL C00369 BC00369 V=100.0  +MOVJ EC00369
MOVL C00370 BC00370 V=400.0  +MOVJ EC00370 VJ=100.00
MOVL C00371 BC00371 V=1000.0  +MOVJ EC00371 VJ=100.00
'Path S3365
SSFTOF
MOVJ C00372 BC00372 VJ=100.00  +MOVJ EC00372 VJ=100.00
MOVL C00373 BC00373 V=400.0  +MOVJ EC00373 VJ=100.00
SMOVL C00374 BC00374 V=100.0  +MOVJ EC00374
SREFP 3 C00375 BC00375  +REFP EC00375
CALL JOB:SEARCH-R1-S1
SET P051 P006
SSFTON P051
SMOVL C00376 BC00376 V=100.0  +MOVJ EC00376
SMOVL C00377 BC00377 V=100.0  +MOVJ EC00377
SREFP 3 C00378 BC00378  +REFP EC00378
CALL JOB:SEARCH-R1-S1
SET P051 P006
SSFTON P051
SMOVL C00379 BC00379 V=100.0  +MOVJ EC00379
MOVL C00380 BC00380 V=400.0  +MOVJ EC00380 VJ=100.00
MOVL C00381 BC00381 V=1000.0  +MOVJ EC00381 VJ=100.00
MOVJ C00382 BC00382 VJ=100.00  +MOVJ EC00382 VJ=100.00
'Path S3366
SSFTOF
MOVJ C00383 BC00383 VJ=100.00  +MOVJ EC00383 VJ=100.00
MOVL C00384 BC00384 V=400.0  +MOVJ EC00384 VJ=100.00
SMOVL C00385 BC00385 V=100.0  +MOVJ EC00385
SREFP 3 C00386 BC00386  +REFP EC00386
CALL JOB:SEARCH-R1-S1
SET P052 P006
SSFTON P052
SMOVL C00387 BC00387 V=100.0  +MOVJ EC00387
SMOVL C00388 BC00388 V=100.0  +MOVJ EC00388
SREFP 3 C00389 BC00389  +REFP EC00389
CALL JOB:SEARCH-R1-S1
SET P052 P006
SSFTON P052
SMOVL C00390 BC00390 V=100.0  +MOVJ EC00390
MOVL C00391 BC00391 V=400.0  +MOVJ EC00391 VJ=100.00
MOVL C00392 BC00392 V=1000.0  +MOVJ EC00392 VJ=100.00
'Path S3367
SSFTOF
MOVJ C00393 BC00393 VJ=100.00  +MOVJ EC00393 VJ=100.00
MOVL C00394 BC00394 V=400.0  +MOVJ EC00394 VJ=100.00
SMOVL C00395 BC00395 V=100.0  +MOVJ EC00395
SREFP 3 C00396 BC00396  +REFP EC00396
CALL JOB:SEARCH-R1-S1
SET P053 P006
SSFTON P053
SMOVL C00397 BC00397 V=100.0  +MOVJ EC00397
SMOVL C00398 BC00398 V=100.0  +MOVJ EC00398
SREFP 3 C00399 BC00399  +REFP EC00399
CALL JOB:SEARCH-R1-S1
SET P053 P006
SSFTON P053
SMOVL C00400 BC00400 V=100.0  +MOVJ EC00400
MOVL C00401 BC00401 V=400.0  +MOVJ EC00401 VJ=100.00
MOVL C00402 BC00402 V=1000.0  +MOVJ EC00402 VJ=100.00
'
'Path W3331
SSFTOF
SSFTON P051
MOVJ C00403 BC00403 VJ=100.00  +MOVJ EC00403 VJ=100.00
SMOVL C00404 BC00404 V=400.0  +MOVJ EC00404
SMOVL C00405 BC00405 V=150.0 PL=0  +MOVJ EC00405
SREFP 1 C00406 BC00406  +REFP EC00406
SREFP 2 C00407 BC00407  +REFP EC00407
MACRO1 MJ#(0) ARGF0
ARCON
SSFTON P050
SMOVL C00408 BC00408 V=10.0  +MOVJ EC00408
SMOVL C00409 BC00409 V=10.0  +MOVJ EC00409
ARCOF
SMOVL C00410 BC00410 V=400.0  +MOVJ EC00410
SMOVL C00411 BC00411 V=1000.0  +MOVJ EC00411
SSFTOF
MOVJ C00412 BC00412 VJ=100.00  +MOVJ EC00412 VJ=100.00
'
'Path W3335
SSFTOF
SSFTON P052
MOVJ C00413 BC00413 VJ=100.00  +MOVJ EC00413 VJ=100.00
SMOVL C00414 BC00414 V=400.0  +MOVJ EC00414
SMOVL C00415 BC00415 V=150.0 PL=0  +MOVJ EC00415
SREFP 1 C00416 BC00416  +REFP EC00416
SREFP 2 C00417 BC00417  +REFP EC00417
MACRO1 MJ#(0) ARGF0
ARCON
SSFTON P053
SMOVL C00418 BC00418 V=10.0  +MOVJ EC00418
ARCOF
SMOVL C00419 BC00419 V=400.0  +MOVJ EC00419
SMOVL C00420 BC00420 V=1000.0  +MOVJ EC00420
SSFTOF
'
'Path W3326
SSFTOF
SSFTON P047
MOVJ C00421 BC00421 VJ=100.00  +MOVJ EC00421 VJ=100.00
SMOVL C00422 BC00422 V=400.0  +MOVJ EC00422
SMOVL C00423 BC00423 V=150.0 PL=0  +MOVJ EC00423
SREFP 1 C00424 BC00424  +REFP EC00424
SREFP 2 C00425 BC00425  +REFP EC00425
MACRO1 MJ#(0) ARGF0
ARCON
SMOVL C00426 BC00426 V=10.0  +MOVJ EC00426
SMOVL C00427 BC00427 V=10.0  +MOVJ EC00427
SMOVL C00428 BC00428 V=10.0  +MOVJ EC00428
ARCOF
SMOVL C00429 BC00429 V=400.0  +MOVJ EC00429
SMOVL C00430 BC00430 V=1000.0  +MOVJ EC00430
SSFTOF
'Path W3327
SSFTOF
SSFTON P048
MOVJ C00431 BC00431 VJ=100.00  +MOVJ EC00431 VJ=100.00
SMOVL C00432 BC00432 V=400.0  +MOVJ EC00432
SMOVL C00433 BC00433 V=150.0 PL=0  +MOVJ EC00433
SREFP 1 C00434 BC00434  +REFP EC00434
SREFP 2 C00435 BC00435  +REFP EC00435
MACRO1 MJ#(0) ARGF0
ARCON
SMOVL C00436 BC00436 V=10.0  +MOVJ EC00436
SMOVL C00437 BC00437 V=10.0  +MOVJ EC00437
SMOVL C00438 BC00438 V=10.0  +MOVJ EC00438
ARCOF
SMOVL C00439 BC00439 V=400.0  +MOVJ EC00439
SMOVL C00440 BC00440 V=1000.0  +MOVJ EC00440
SSFTOF
'Path W3328
SSFTOF
SSFTON P049
MOVJ C00441 BC00441 VJ=100.00  +MOVJ EC00441 VJ=100.00
SMOVL C00442 BC00442 V=400.0  +MOVJ EC00442
SMOVL C00443 BC00443 V=150.0 PL=0  +MOVJ EC00443
SREFP 1 C00444 BC00444  +REFP EC00444
SREFP 2 C00445 BC00445  +REFP EC00445
MACRO1 MJ#(0) ARGF0
ARCON
SMOVL C00446 BC00446 V=10.0  +MOVJ EC00446
SMOVL C00447 BC00447 V=10.0  +MOVJ EC00447
SMOVL C00448 BC00448 V=10.0  +MOVJ EC00448
ARCOF
SMOVL C00449 BC00449 V=400.0  +MOVJ EC00449
SMOVL C00450 BC00450 V=1000.0  +MOVJ EC00450
SSFTOF
MOVJ C00451 BC00451 VJ=100.00  +MOVJ EC00451 VJ=100.00
'
'Path W3323
SSFTOF
SSFTON P044
MOVJ C00452 BC00452 VJ=100.00  +MOVJ EC00452 VJ=100.00
SMOVL C00453 BC00453 V=400.0  +MOVJ EC00453
SMOVL C00454 BC00454 V=150.0 PL=0  +MOVJ EC00454
SREFP 1 C00455 BC00455  +REFP EC00455
SREFP 2 C00456 BC00456  +REFP EC00456
MACRO1 MJ#(0) ARGF0
ARCON
SMOVL C00457 BC00457 V=10.0  +MOVJ EC00457
SMOVL C00458 BC00458 V=10.0  +MOVJ EC00458
SMOVL C00459 BC00459 V=10.0  +MOVJ EC00459
ARCOF
SMOVL C00460 BC00460 V=400.0  +MOVJ EC00460
SMOVL C00461 BC00461 V=1000.0  +MOVJ EC00461
SSFTOF
'Path W3324
SSFTOF
SSFTON P045
MOVJ C00462 BC00462 VJ=100.00  +MOVJ EC00462 VJ=100.00
SMOVL C00463 BC00463 V=400.0  +MOVJ EC00463
SMOVL C00464 BC00464 V=150.0 PL=0  +MOVJ EC00464
SREFP 1 C00465 BC00465  +REFP EC00465
SREFP 2 C00466 BC00466  +REFP EC00466
MACRO1 MJ#(0) ARGF0
ARCON
SMOVL C00467 BC00467 V=10.0  +MOVJ EC00467
SMOVL C00468 BC00468 V=10.0  +MOVJ EC00468
SMOVL C00469 BC00469 V=10.0  +MOVJ EC00469
ARCOF
SMOVL C00470 BC00470 V=400.0  +MOVJ EC00470
SMOVL C00471 BC00471 V=1000.0  +MOVJ EC00471
SSFTOF
'Path W3325
SSFTOF
SSFTON P046
MOVJ C00472 BC00472 VJ=100.00  +MOVJ EC00472 VJ=100.00
SMOVL C00473 BC00473 V=400.0  +MOVJ EC00473
SMOVL C00474 BC00474 V=150.0 PL=0  +MOVJ EC00474
SREFP 1 C00475 BC00475  +REFP EC00475
SREFP 2 C00476 BC00476  +REFP EC00476
MACRO1 MJ#(0) ARGF0
ARCON
SMOVL C00477 BC00477 V=10.0  +MOVJ EC00477
SMOVL C00478 BC00478 V=10.0  +MOVJ EC00478
SMOVL C00479 BC00479 V=10.0  +MOVJ EC00479
ARCOF
SMOVL C00480 BC00480 V=400.0  +MOVJ EC00480
SMOVL C00481 BC00481 V=1000.0  +MOVJ EC00481
SSFTOF
MOVJ C00482 BC00482 VJ=100.00  +MOVJ EC00482 VJ=100.00
'
'
'Path W3320
SSFTOF
SSFTON P041
MOVJ C00483 BC00483 VJ=100.00  +MOVJ EC00483 VJ=100.00
SMOVL C00484 BC00484 V=400.0  +MOVJ EC00484
SMOVL C00485 BC00485 V=100.0 PL=0  +MOVJ EC00485
SREFP 1 C00486 BC00486  +REFP EC00486
SREFP 2 C00487 BC00487  +REFP EC00487
MACRO1 MJ#(0) ARGF0
ARCON
SMOVL C00488 BC00488 V=10.0  +MOVJ EC00488
SMOVL C00489 BC00489 V=10.0  +MOVJ EC00489
SMOVL C00490 BC00490 V=10.0  +MOVJ EC00490
ARCOF
SMOVL C00491 BC00491 V=400.0  +MOVJ EC00491
SMOVL C00492 BC00492 V=1000.0  +MOVJ EC00492
SSFTOF
'Path W3321
SSFTOF
SSFTON P042
MOVJ C00493 BC00493 VJ=100.00  +MOVJ EC00493 VJ=100.00
SMOVL C00494 BC00494 V=400.0  +MOVJ EC00494
SMOVL C00495 BC00495 V=100.0 PL=0  +MOVJ EC00495
SREFP 1 C00496 BC00496  +REFP EC00496
SREFP 2 C00497 BC00497  +REFP EC00497
MACRO1 MJ#(0) ARGF0
ARCON
SMOVL C00498 BC00498 V=10.0  +MOVJ EC00498
SMOVL C00499 BC00499 V=10.0  +MOVJ EC00499
SMOVL C00500 BC00500 V=10.0  +MOVJ EC00500
ARCOF
SMOVL C00501 BC00501 V=400.0  +MOVJ EC00501
SMOVL C00502 BC00502 V=1000.0  +MOVJ EC00502
SSFTOF
'Path W3322
SSFTOF
SSFTON P043
MOVJ C00503 BC00503 VJ=100.00  +MOVJ EC00503 VJ=100.00
SMOVL C00504 BC00504 V=400.0  +MOVJ EC00504
SMOVL C00505 BC00505 V=100.0 PL=0  +MOVJ EC00505
SREFP 1 C00506 BC00506  +REFP EC00506
SREFP 2 C00507 BC00507  +REFP EC00507
MACRO1 MJ#(0) ARGF0
ARCON
SMOVL C00508 BC00508 V=10.0  +MOVJ EC00508
SMOVL C00509 BC00509 V=10.0  +MOVJ EC00509
SMOVL C00510 BC00510 V=10.0  +MOVJ EC00510
ARCOF
SMOVL C00511 BC00511 V=400.0  +MOVJ EC00511
SMOVL C00512 BC00512 V=1000.0  +MOVJ EC00512
SSFTOF
MOVJ C00513 BC00513 VJ=100.00  +MOVJ EC00513 VJ=100.00
MOVJ C00514 BC00514 VJ=100.00  +MOVJ EC00514 VJ=100.00
END
